fb_eib_kabinetFloorHeatingPowerSpRec(
	strData_Rec := fb_KL6301_0.str_Data_Rec,
	Group_Address := kabinetFloorHeatingPowerSp_adr,
	iData => kabinetFloorHeatingSp
	);
data2floor[103] := INT_TO_BYTE(kabinetFloorHeatingSp);

fb_eib_studioFloorHeatingPowerSpRec(
	strData_Rec := fb_KL6301_0.str_Data_Rec,
	Group_Address := studioFloorHeatingPowerSp_adr,
	iData => studioFloorHeatingSp
	);
data2floor[104] := INT_TO_BYTE(studioFloorHeatingSp);

fb_balkon_peryla_read(strData_Rec:=fb_KL6301_0.str_Data_Rec,   Group_Address:=balkon_peryla_adr);
IF NOT  fb_balkon_peryla_read.bDataReceive OR NOT fb_eib_twillight_rec.bDataReceive  THEN
	data2floor[100].0:= fb_balkon_peryla_read.bdata OR  fb_eib_twillight_rec.bData ;
END_IF
fb_kino_l_read(strData_Rec:=fb_KL6301_0.str_Data_Rec,   Group_Address:=kino_l_adr);
IF NOT  fb_kino_l_read.bDataReceive THEN
	data2floor[100].1:= fb_kino_l_read.bdata;
END_IF
fb_balkon_bra_read(strData_Rec:=fb_KL6301_0.str_Data_Rec,   Group_Address:=balkon_bra_adr);
IF NOT  fb_balkon_bra_read.bDataReceive OR NOT fb_eib_twillight_rec.bDataReceive THEN
	data2floor[100].2:= fb_balkon_bra_read.bdata OR fb_eib_twillight_rec.bData;
END_IF
fb_kabinet_balkon_l_read(strData_Rec:=fb_KL6301_0.str_Data_Rec,   Group_Address:=kabinet_balkon_l_adr);
IF NOT  fb_kabinet_balkon_l_read.bDataReceive THEN
	data2floor[100].3:= fb_kabinet_balkon_l_read.bdata;
END_IF
fb_balkon_read(strData_Rec:=fb_KL6301_0.str_Data_Rec,   Group_Address:=balkon_adr);
IF NOT  fb_balkon_read.bDataReceive THEN
	data2floor[100].4:= fb_balkon_read.bdata;
END_IF
fb_korydor1_read(strData_Rec:=fb_KL6301_0.str_Data_Rec,   Group_Address:=korydor1_adr);
IF NOT  fb_korydor1_read.bDataReceive THEN
	data2floor[100].5:= fb_korydor1_read.bdata;
END_IF
fb_kino_bra_read(strData_Rec:=fb_KL6301_0.str_Data_Rec,   Group_Address:=kino_bra_adr);
IF NOT  fb_kino_bra_read.bDataReceive THEN
	data2floor[100].6:= fb_kino_bra_read.bdata;
END_IF
fb_studio_pidsvitka_read(strData_Rec:=fb_KL6301_0.str_Data_Rec,   Group_Address:=studio_pidsvitka_adr);
IF NOT  fb_studio_pidsvitka_read.bDataReceive THEN
	data2floor[100].7:= fb_studio_pidsvitka_read.bdata;
END_IF
fb_skhody2_3_read(strData_Rec:=fb_KL6301_0.str_Data_Rec,   Group_Address:=skhody2_3_adr);
IF NOT  fb_skhody2_3_read.bDataReceive THEN
	data2floor[101].0:= fb_skhody2_3_read.bdata;
END_IF
fb_studio_l_read(strData_Rec:=fb_KL6301_0.str_Data_Rec,   Group_Address:=studio_l_adr);
IF NOT  fb_studio_l_read.bDataReceive THEN
	data2floor[101].1:= fb_studio_l_read.bdata;
END_IF
fb_kabinet_svitlo_read(strData_Rec:=fb_KL6301_0.str_Data_Rec,   Group_Address:=kabinet_svitlo_adr);
IF NOT  fb_kabinet_svitlo_read.bDataReceive THEN
	data2floor[101].2:= fb_kabinet_svitlo_read.bdata;
END_IF
fb_kabinet_kobra_read(strData_Rec:=fb_KL6301_0.str_Data_Rec,   Group_Address:=kabinet_kobra_adr);
IF NOT  fb_kabinet_kobra_read.bDataReceive THEN
	data2floor[101].3:= fb_kabinet_kobra_read.bdata;
END_IF
fb_tambur2_read(strData_Rec:=fb_KL6301_0.str_Data_Rec,   Group_Address:=tambur2_adr);
IF NOT  fb_tambur2_read.bDataReceive THEN
	data2floor[101].4:= fb_tambur2_read.bdata;
END_IF
fb_stend_read(strData_Rec:=fb_KL6301_0.str_Data_Rec,   Group_Address:=stend_adr);
IF NOT  fb_stend_read.bDataReceive THEN
	data2floor[101].5:= fb_stend_read.bdata;
END_IF
fb_skhody_peryla_read(strData_Rec:=fb_KL6301_0.str_Data_Rec,   Group_Address:=skhody_peryla_adr);
IF NOT  fb_skhody_peryla_read.bDataReceive OR NOT  fb_eib_twillight_rec.bDataReceive THEN
	data2floor[101].6:= fb_skhody_peryla_read.bdata OR  fb_eib_twillight_rec.bData;
END_IF

fb_kino_bra_dim_read(strData_Rec:=fb_KL6301_0.str_Data_Rec,   Group_Address:=kino_bra_dimming_adr);
IF NOT  fb_kino_bra_dim_read.bDataReceive THEN
	data2floor[102]:= INT_TO_BYTE(fb_kino_bra_dim_read.iData);
END_IF


(*sending*)
fb_balkon_peryla_send_status_ex(imode:=eib_send_mode_floor2, bStart:=eib_send_cyclical_start_floor2, str_Rec:=fb_KL6301_0.str_Data_Rec, bData:=balkon_peryla,  Group_Address:=balkon_peryla_status_adr);
fb_kino_l_send_status_ex(imode:=eib_send_mode_floor2, bStart:=eib_send_cyclical_start_floor2, str_Rec:=fb_KL6301_0.str_Data_Rec, bData:=kino_l,  Group_Address:=kino_l_status_adr);
fb_balkon_bra_send_status_ex(imode:=eib_send_mode_floor2, bStart:=eib_send_cyclical_start_floor2, str_Rec:=fb_KL6301_0.str_Data_Rec, bData:=balkon_bra,  Group_Address:=balkon_bra_status_adr);
fb_kabinet_balkon_l_send_status_ex(imode:=eib_send_mode_floor2, bStart:=eib_send_cyclical_start_floor2, str_Rec:=fb_KL6301_0.str_Data_Rec, bData:=kabinet_balkon_l,  Group_Address:=kabinet_balkon_l_status_adr);
fb_balkon_send_status_ex(imode:=eib_send_mode_floor2, bStart:=eib_send_cyclical_start_floor2, str_Rec:=fb_KL6301_0.str_Data_Rec, bData:=balkon,  Group_Address:=balkon_status_adr);
fb_korydor1_send_status_ex(imode:=eib_send_mode_floor2, bStart:=eib_send_cyclical_start_floor2, str_Rec:=fb_KL6301_0.str_Data_Rec, bData:=korydor1,  Group_Address:=korydor1_status_adr);
fb_kino_bra_send_status_ex(imode:=eib_send_mode_floor2, bStart:=eib_send_cyclical_start_floor2, str_Rec:=fb_KL6301_0.str_Data_Rec, bData:=kino_bra,  Group_Address:=kino_bra_status_adr);
fb_studio_pidsvitka_send_status_ex(imode:=eib_send_mode_floor2, bStart:=eib_send_cyclical_start_floor2, str_Rec:=fb_KL6301_0.str_Data_Rec, bData:=studio_pidsvitka,  Group_Address:=studio_pidsvitka_status_adr);
fb_skhody2_3_send_status_ex(imode:=eib_send_mode_floor2, bStart:=eib_send_cyclical_start_floor2, str_Rec:=fb_KL6301_0.str_Data_Rec, bData:=skhody2_3,  Group_Address:=skhody2_3_status_adr);
fb_studio_l_send_status_ex(imode:=eib_send_mode_floor2, bStart:=eib_send_cyclical_start_floor2, str_Rec:=fb_KL6301_0.str_Data_Rec, bData:=studio_l,  Group_Address:=studio_l_status_adr);
fb_kabinet_svitlo_send_status_ex(imode:=eib_send_mode_floor2, bStart:=eib_send_cyclical_start_floor2, str_Rec:=fb_KL6301_0.str_Data_Rec, bData:=kabinet_svitlo,  Group_Address:=kabinet_svitlo_status_adr);
fb_kabinet_kobra_send_status_ex(imode:=eib_send_mode_floor2, bStart:=eib_send_cyclical_start_floor2, str_Rec:=fb_KL6301_0.str_Data_Rec, bData:=kabinet_kobra,  Group_Address:=kabinet_kobra_status_adr);
fb_tambur2_send_status_ex(imode:=eib_send_mode_floor2, bStart:=eib_send_cyclical_start_floor2, str_Rec:=fb_KL6301_0.str_Data_Rec, bData:=tambur2,  Group_Address:=tambur2_status_adr);
fb_stend_send_status_ex(imode:=eib_send_mode_floor2, bStart:=eib_send_cyclical_start_floor2, str_Rec:=fb_KL6301_0.str_Data_Rec, bData:=stend,  Group_Address:=stend_status_adr);
fb_skhody_peryla_send_status_ex(imode:=eib_send_mode_floor2, bStart:=eib_send_cyclical_start_floor2, str_Rec:=fb_KL6301_0.str_Data_Rec, bData:=skhody_peryla,  Group_Address:=skhody_peryla_status_adr);
fb_kino_bra_send_dim_status_ex(imode:=eib_send_mode_floor2, bstart:=eib_send_cyclical_start_floor2, str_Rec:=fb_KL6301_0.str_Data_Rec, idata:=BYTE_TO_INT(kino_bra_dim_value) );


IF fb_balkon_peryla_send_status_ex.bBusy THEN
	data2floor[100].0:=balkon_peryla;
END_IF
IF fb_kino_l_send_status_ex.bBusy OR fb_heartbeat_timer.Q THEN
	data2floor[100].1:=kino_l;
END_IF
IF fb_balkon_bra_send_status_ex.bBusy OR fb_heartbeat_timer.Q THEN
	data2floor[100].2:=balkon_bra;
END_IF
IF fb_kabinet_balkon_l_send_status_ex.bBusy OR fb_heartbeat_timer.Q THEN
	data2floor[100].3:=kabinet_balkon_l;
END_IF
IF fb_balkon_send_status_ex.bBusy OR fb_heartbeat_timer.Q THEN
	data2floor[100].4:=balkon;
END_IF
IF fb_korydor1_send_status_ex.bBusy OR fb_heartbeat_timer.Q THEN
	data2floor[100].5:=korydor1;
END_IF
IF fb_kino_bra_send_status_ex.bBusy OR fb_heartbeat_timer.Q THEN
	data2floor[100].6:=kino_bra;
END_IF
IF fb_studio_pidsvitka_send_status_ex.bBusy OR fb_heartbeat_timer.Q THEN
	data2floor[100].7:=studio_pidsvitka;
END_IF
IF fb_skhody2_3_send_status_ex.bBusy OR fb_heartbeat_timer.Q THEN
	data2floor[101].0:=skhody2_3;
END_IF
IF fb_studio_l_send_status_ex.bBusy OR fb_heartbeat_timer.Q THEN
	data2floor[101].1:=studio_l;
END_IF
IF fb_kabinet_svitlo_send_status_ex.bBusy OR fb_heartbeat_timer.Q THEN
	data2floor[101].2:=kabinet_svitlo;
END_IF
IF fb_kabinet_kobra_send_status_ex.bBusy OR fb_heartbeat_timer.Q THEN
	data2floor[101].3:=kabinet_kobra;
END_IF
IF fb_tambur2_send_status_ex.bBusy OR fb_heartbeat_timer.Q THEN
	data2floor[101].4:=tambur2;
END_IF
IF fb_stend_send_status_ex.bBusy OR fb_heartbeat_timer.Q THEN
	data2floor[101].5:=stend;
END_IF
IF fb_skhody_peryla_send_status_ex.bBusy OR fb_heartbeat_timer.Q THEN
	data2floor[101].6:=skhody_peryla;
END_IF
IF fb_kino_bra_send_dim_status_ex.bBusy THEN
	data2floor[102]:=INT_TO_BYTE(kino_bra_dim_value);
END_IF
END_ACTION
ACTION floor3:
(*read*)
fb_spalnya_kontrazhury_read(
	strData_Rec := fb_KL6301_0.str_Data_Rec,
	Group_Address := spalnya_kontrazhury_adr,
	bData => eib_spalnya_kontrazhury
	);

fb_spalnya_balkon_read(
	strData_Rec := fb_KL6301_0.str_Data_Rec,
	Group_Address := spalnya_balkon_adr,
	bData => eib_spalnya_balkon
	);

fb_spalnya_kulbaba_read(
	strData_Rec := fb_KL6301_0.str_Data_Rec,
	Group_Address := spalnya_kulbaba_adr,
	bData => eib_spalnya_kulbaba
	);

fb_eib_su3FloorHeatingPowerSpRec(
	strData_Rec := fb_KL6301_0.str_Data_Rec,
	Group_Address := su3FloorHeatingPowerSp_adr,
	iData => su3FloorHeatingSp
	);

fb_eib_freshbarFloorHeatingPowerSpRec(
	strData_Rec := fb_KL6301_0.str_Data_Rec,
	Group_Address := freshbarFloorHeatingPowerSp_adr,
	iData => freshbarFloorHeatingSp
	);

fb_eib_servernaFloorHeatingPowerSpRec(
	strData_Rec := fb_KL6301_0.str_Data_Rec,
	Group_Address := servernaFloorHeatingPowerSp_adr,
	iData => servernaFloorHeatingSp
	);

fb_eib_spalnyaFloorHeatingPowerSpRec(
	strData_Rec := fb_KL6301_0.str_Data_Rec,
	Group_Address := spalnyaFloorHeatingPowerSp_adr,
	iData => spalnyaFloorHeatingSp
	);

fb_eib_dytjachaFloorHeatingPowerSpRec(
	strData_Rec := fb_KL6301_0.str_Data_Rec,
	Group_Address := dytjachaFloorHeatingPowerSp_adr,
	iData => dytjachaFloorHeatingSp
	);

(*
fb_spalnya_kontrazhur_b_read(strData_Rec:=fb_KL6301_0.str_Data_Rec, Group_Address:=spalnya_kontrazhur_b_adr);
fb_spalnya_kontrazhur_l_read(strData_Rec:=fb_KL6301_0.str_Data_Rec, Group_Address:=spalnya_kontrazhur_l_adr);
*)
fb_su3_stina_read(
	strData_Rec := fb_KL6301_0.str_Data_Rec,
	Group_Address := su3_stina_adr,
	bData => eib_su3_stina
	);

fb_su3_pidsvitka_read(
	strData_Rec := fb_KL6301_0.str_Data_Rec,
	Group_Address := su3_pidsvitka_adr,
	bData => eib_su3_pidsvitka
	);

fb_su3_bra_read(
	strData_Rec := fb_KL6301_0.str_Data_Rec,
	Group_Address := su3_bra_adr,
	bData => eib_su3_bra
	);

fb_su3_kontrazhur_read(
	strData_Rec := fb_KL6301_0.str_Data_Rec,
	Group_Address := su3_kontrazhury_adr,
	bData => eib_su3_kontrazhury
	);

fb_su3_vent_read(
	strData_Rec := fb_KL6301_0.str_Data_Rec,
	Group_Address := su3_vent_adr,
	bData => eib_su3_vent
	);

fb_su3_lampa_read(
	strData_Rec := fb_KL6301_0.str_Data_Rec,
	Group_Address := su3_lampa_adr,
	bData => eib_su3_lampa
	);

fb_dytjacha_read(
	strData_Rec := fb_KL6301_0.str_Data_Rec,
	Group_Address := dytjacha_adr,
	bData => eib_dytjacha
	);

fb_dytjacha_bra_read(
	strData_Rec := fb_KL6301_0.str_Data_Rec,
	Group_Address := dytjacha_bra_adr,
	bData => eib_dytjacha_bra
	);

fb_garderob_read(
	strData_Rec := fb_KL6301_0.str_Data_Rec,
	Group_Address := garderob_adr,
	bData => eib_garderob
	);

fb_bar_read(
	strData_Rec := fb_KL6301_0.str_Data_Rec,
	Group_Address := bar_adr,
	bData => eib_bar
	);

fb_korydor_skeli_read(
	strData_Rec := fb_KL6301_0.str_Data_Rec,
	Group_Address := korydor_skeli_adr,
	bData => eib_korydor_skeli
	);

fb_choven_read(
	strData_Rec := fb_KL6301_0.str_Data_Rec,
	Group_Address := choven_adr,
	bData => eib_choven
	);

fb_korydor_lampa_read(
	strData_Rec := fb_KL6301_0.str_Data_Rec,
	Group_Address := korydor_lampa_adr,
	bData => eib_korydor_lampa
	);

fb_serverna_read(
	strData_Rec := fb_KL6301_0.str_Data_Rec,
	Group_Address := serverna_adr,
	bData => eib_serverna
	);

fb_korydor_svitlo_read(
	strData_Rec := fb_KL6301_0.str_Data_Rec,
	Group_Address := korydor_svitlo_adr,
	bData => eib_korydor_svitlo
	);

(*sending*)
(*
fb_spalnya_kontrazhur_b_send_status_ex(imode:=eib_send_mode_floor3, bStart:=eib_send_cyclical_start_floor3, str_Rec:=fb_KL6301_0.str_Data_Rec, Group_Address:=spalnya_kontrazhur_b_status_adr, bData:=spalnya_kontrazhur_b);
fb_spalnya_kontrazhur_l_send_status_ex(imode:=eib_send_mode_floor3, bStart:=eib_send_cyclical_start_floor3, str_Rec:=fb_KL6301_0.str_Data_Rec, Group_Address:=spalnya_kontrazhur_l_status_adr, bData:=spalnya_kontrazhur_l);

*)
fb_su3_stina_send_status_ex(
	imode := eib_send_mode_floor3,
	bStart := eib_send_cyclical_start_floor3,
	str_Rec := fb_KL6301_0.str_Data_Rec,
	Group_Address := su3_stina_status_adr,
	bData := su3_stina
	);

fb_su3_pidsvitka_send_status_ex(
	imode := eib_send_mode_floor3,
	bStart := eib_send_cyclical_start_floor3,
	str_Rec := fb_KL6301_0.str_Data_Rec,
	Group_Address := su3_pidsvitka_status_adr,
	bData := su3_pidsvitka
	);

fb_su3_bra_send_status_ex(
	imode := eib_send_mode_floor3,
	bStart := eib_send_cyclical_start_floor3,
	str_Rec := fb_KL6301_0.str_Data_Rec,
	Group_Address := su3_bra_status_adr,
	bData := su3_bra
	);

fb_su3_kontrazhur_send_status_ex(
	imode := eib_send_mode_floor3,
	bStart := eib_send_cyclical_start_floor3,
	str_Rec := fb_KL6301_0.str_Data_Rec,
	Group_Address := su3_kontrazhury_status_adr,
	bData := su3_kontrazhur
	);

fb_su3_vent_send_status_ex(
	imode := eib_send_mode_floor3,
	bStart := eib_send_cyclical_start_floor3,
	str_Rec := fb_KL6301_0.str_Data_Rec,
	Group_Address := su3_vent_status_adr,
	bData := su3_vent
	);

fb_su3_lampa_send_status_ex(
	imode := eib_send_mode_floor3,
	bStart := eib_send_cyclical_start_floor3,
	str_Rec := fb_KL6301_0.str_Data_Rec,
	Group_Address := su3_lampa_status_adr,
	bData := su3_lampa
	);

fb_dytjacha_send_status_ex(
	imode := eib_send_mode_floor3,
	bStart := eib_send_cyclical_start_floor3,
	str_Rec := fb_KL6301_0.str_Data_Rec,
	Group_Address := dytjacha_status_adr,
	bData := dytjacha
	);

fb_dytjacha_bra_send_status_ex(
	imode := eib_send_mode_floor3,
	bStart := eib_send_cyclical_start_floor3,
	str_Rec := fb_KL6301_0.str_Data_Rec,
	Group_Address := dytjacha_bra_status_adr,
	bData := dytjacha_bra
	);

fb_garderob_send_status_ex(
	imode := eib_send_mode_floor3,
	bStart := eib_send_cyclical_start_floor3,
	str_Rec := fb_KL6301_0.str_Data_Rec,
	Group_Address := garderob_status_adr,
	bData := garderob
	);

fb_bar_send_status_ex(
	imode := eib_send_mode_floor3,
	bStart := eib_send_cyclical_start_floor3,
	str_Rec := fb_KL6301_0.str_Data_Rec,
	Group_Address := bar_status_adr,
	bData := bar
	);

fb_korydor_skeli_send_status_ex(
	imode := eib_send_mode_floor3,
	bStart := eib_send_cyclical_start_floor3,
	str_Rec := fb_KL6301_0.str_Data_Rec,
	Group_Address := korydor_skeli_status_adr,
	bData := korydor_skeli
	);

fb_choven_send_status_ex(
	imode := eib_send_mode_floor3,
	bStart := eib_send_cyclical_start_floor3,
	str_Rec := fb_KL6301_0.str_Data_Rec,
	Group_Address := choven_status_adr,
	bData := choven
	);

fb_korydor_lampa_send_status_ex(
	imode := eib_send_mode_floor3,
	bStart := eib_send_cyclical_start_floor3,
	str_Rec := fb_KL6301_0.str_Data_Rec,
	Group_Address := korydor_lampa_status_adr,
	bData := korydor_lampa
	);

fb_serverna_send_status_ex(
	imode := eib_send_mode_floor3,
	bStart := eib_send_cyclical_start_floor3,
	str_Rec := fb_KL6301_0.str_Data_Rec,
	Group_Address := serverna_status_adr,
	bData := serverna
	);

fb_korydor_svitlo_send_status_ex(
	imode := eib_send_mode_floor3,
	bStart := eib_send_cyclical_start_floor3,
	str_Rec := fb_KL6301_0.str_Data_Rec,
	Group_Address := korydor_svitlo_status_adr,
	bData := korydor_svitlo
	);

fb_spalnya_balkon_send_status_ex(
	imode := eib_send_mode_floor3,
	bStart := eib_send_cyclical_start_floor3,
	str_Rec := fb_KL6301_0.str_Data_Rec,
	Group_Address := spalnya_balkon_status_adr,
	bData := spalnya_balkon
	);

fb_spalnya_kulbaba_send_status_ex(
	imode := eib_send_mode_floor3,
	bStart := eib_send_cyclical_start_floor3,
	str_Rec := fb_KL6301_0.str_Data_Rec,
	Group_Address := spalnya_kulbaba_status_adr,
	bData := spalnya_kulbaba
	);

fb_spalnya_kontrazhury_send_status_ex(
	imode := eib_send_mode_floor3,
	bStart := eib_send_cyclical_start_floor3,
	str_Rec := fb_KL6301_0.str_Data_Rec,
	Group_Address := spalnya_kontrazhury_status_adr,
	bData :=spalnya_kontrazhur
	);

fb_spalnya_lift_send_status_ex(
	imode := eib_send_mode_floor3,
	bStart := eib_send_cyclical_start_floor3,
	str_Rec := fb_KL6301_0.str_Data_Rec,
	Group_Address := lift_spalnya_status_EIB_addr,
	bData := eib_lift_spalnya_move
	);
END_ACTION
ACTION gym_and_outside:
data_gym[0].0:=bDarkOutside OR b_eib_twillight;
data_gym[0].1:=1;

data_gym[1]:=WORD_TO_BYTE(system_time.wHour);
data_gym[3]:=WORD_TO_BYTE(system_time.wMinute);

MEMCPY(ADR(data_gym[6] ), ADR(OAT), SIZEOF(OAT));


fb_outside_bigBulbs_read(strData_Rec:=fb_KL6301_0.str_Data_Rec, Group_Address:=outside_bigBulbs_adr );
IF NOT  fb_outside_Bigbulbs_read.bDataReceive THEN
	data_gym[12].3:= fb_outside_bigBulbs_read.bdata;
END_IF

fb_outside_pingPongTable_read(strData_Rec:=fb_KL6301_0.str_Data_Rec, Group_Address:=outside_pingPongTable_adr );
IF NOT  fb_outside_pingPongTable_read.bDataReceive THEN
	data_gym[12].4:= fb_outside_pingPongTable_read.bdata;
END_IF
fb_outside_plantsLightning_read(strData_Rec:=fb_KL6301_0.str_Data_Rec, Group_Address:=outside_plantsLightning_adr );
IF NOT  fb_outside_plantsLightning_read.bDataReceive THEN
	data_gym[12].5:= fb_outside_plantsLightning_read.bdata;
END_IF

fb_outside_smallBulbs_read(strData_Rec:=fb_KL6301_0.str_Data_Rec, Group_Address:=outside_smallBulbs_adr );
IF NOT  fb_outside_smallBulbs_read.bDataReceive THEN
	data_gym[12].6:= fb_outside_smallBulbs_read.bdata;
END_IF


(*sending*)


fb_outside_bigBulbs_send_status_ex(imode:=eib_send_mode_floor4, bStart:=eib_send_cyclical_start_floor4, str_Rec:=fb_KL6301_0.str_Data_Rec, bData:=outside_bigBulbs,  Group_Address:=outside_bigBulbs_status_adr);
fb_outside_pingPongTable_send_status_ex(imode:=eib_send_mode_floor4, bStart:=eib_send_cyclical_start_floor4, str_Rec:=fb_KL6301_0.str_Data_Rec, bData:=outside_pingPongTable,  Group_Address:=outside_pingPongTable_status_adr);
fb_outside_plantsLightning_send_status_ex(imode:=eib_send_mode_floor4, bStart:=eib_send_cyclical_start_floor4, str_Rec:=fb_KL6301_0.str_Data_Rec, bData:=outside_plantsLightning,  Group_Address:=outside_plantsLightning_status_adr);
fb_outside_smallBulbs_send_status_ex(imode:=eib_send_mode_floor4, bStart:=eib_send_cyclical_start_floor4, str_Rec:=fb_KL6301_0.str_Data_Rec, bData:=outside_smallBulbs,  Group_Address:=outside_smallBulbs_status_adr);


IF fb_gym_light_send_status_ex.bBusy OR fb_heartbeat_timer.Q  THEN
	data_gym[12].2:=gym_light;
END_IF


IF fb_outside_bigBulbs_send_status_ex.bBusy OR fb_heartbeat_timer.Q  THEN
	data_gym[12].3:=outside_bigBulbs;
END_IF

IF fb_outside_pingPongTable_send_status_ex.bBusy OR fb_heartbeat_timer.Q  THEN
	data_gym[12].4:=outside_pingPongTable;
END_IF

IF fb_outside_plantsLightning_send_status_ex.bBusy OR fb_heartbeat_timer.Q  THEN
	data_gym[12].5:=outside_plantsLightning;
END_IF

IF fb_outside_smallBulbs_send_status_ex.bBusy OR fb_heartbeat_timer.Q  THEN
	data_gym[12].6:=outside_smallBulbs;
END_IF
END_ACTION
ACTION timers:
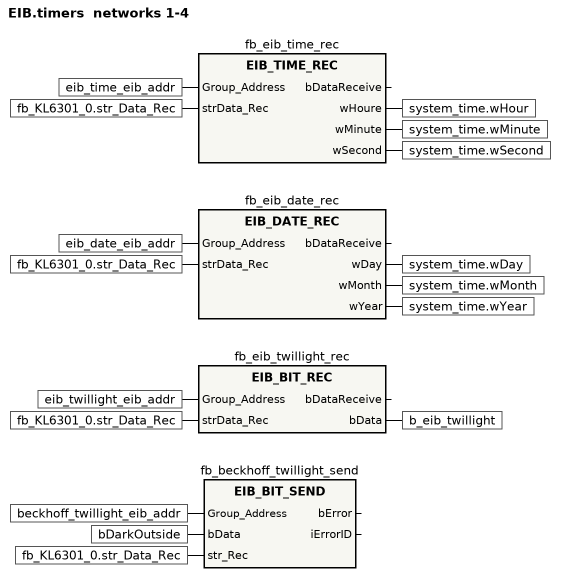
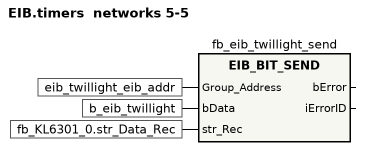
_FBD_ (* Function Block Diagram *)
NETWORK 1
	fb_eib_time_rec:EIB_TIME_REC(Group_Address: eib_time_eib_addr, strData_Rec: fb_KL6301_0.str_Data_Rec, wHoure => system_time.wHour, wMinute => system_time.wMinute, wSecond => system_time.wSecond)
NETWORK 2
	fb_eib_date_rec:EIB_DATE_REC(Group_Address: eib_date_eib_addr, strData_Rec: fb_KL6301_0.str_Data_Rec, wDay => system_time.wDay, wMonth => system_time.wMonth, wYear => system_time.wYear)
NETWORK 3
	fb_eib_twillight_rec:EIB_BIT_REC(Group_Address: eib_twillight_eib_addr, strData_Rec: fb_KL6301_0.str_Data_Rec, bData => b_eib_twillight)
NETWORK 4
	fb_beckhoff_twillight_send:EIB_BIT_SEND(Group_Address: beckhoff_twillight_eib_addr, bData: bDarkOutside, str_Rec: fb_KL6301_0.str_Data_Rec)
NETWORK 5
	fb_eib_twillight_send:EIB_BIT_SEND(Group_Address: eib_twillight_eib_addr, bData: b_eib_twillight, str_Rec: fb_KL6301_0.str_Data_Rec)
_END_FBD_
(* the same logic as Structured Text *)
(* Network 1 *)
fb_eib_time_rec(Group_Address := eib_time_eib_addr, strData_Rec := fb_KL6301_0.str_Data_Rec);
system_time.wHour := fb_eib_time_rec.wHoure;
system_time.wMinute := fb_eib_time_rec.wMinute;
system_time.wSecond := fb_eib_time_rec.wSecond;
(* Network 2 *)
fb_eib_date_rec(Group_Address := eib_date_eib_addr, strData_Rec := fb_KL6301_0.str_Data_Rec);
system_time.wDay := fb_eib_date_rec.wDay;
system_time.wMonth := fb_eib_date_rec.wMonth;
system_time.wYear := fb_eib_date_rec.wYear;
(* Network 3 *)
fb_eib_twillight_rec(Group_Address := eib_twillight_eib_addr, strData_Rec := fb_KL6301_0.str_Data_Rec);
b_eib_twillight := fb_eib_twillight_rec.bData;
(* Network 4 *)
fb_beckhoff_twillight_send(Group_Address := beckhoff_twillight_eib_addr, bData := bDarkOutside, str_Rec := fb_KL6301_0.str_Data_Rec);
(* Network 5 *)
fb_eib_twillight_send(Group_Address := eib_twillight_eib_addr, bData := b_eib_twillight, str_Rec := fb_KL6301_0.str_Data_Rec);
END_ACTION

(* POU RANGE_TO_RANGE, ST *)
FUNCTION RANGE_TO_RANGE : INT
VAR_INPUT
	by_input:BYTE;
	in_low_value: INT;
	in_high_value:INT;
	out_low_value: INT;
	out_high_value:INT;
END_VAR
VAR
	r_res: REAL;
	r_input: REAL;
END_VAR
r_input:=BYTE_TO_REAL(by_input);
IF out_high_value>out_low_value THEN
	r_res:=r_input/(in_high_value - in_low_value)*(out_high_value - out_low_value);
ELSE
	r_res:=out_low_value - (r_input / (in_high_value - in_low_value)*(out_low_value - out_high_value));
END_IF
RANGE_TO_RANGE:=REAL_TO_INT(r_res);
END_FUNCTION

(* POU GREATEST_OF, ST *)
FUNCTION GREATEST_OF : REAL
VAR_INPUT
	r_in1,r_in2:REAL;
END_VAR
VAR
END_VAR
IF r_in1>=r_in2 THEN
	GREATEST_OF:=r_in1;
ELSE
	GREATEST_OF:=r_in2;
END_IF
END_FUNCTION

(* POU Light, CFC *)
PROGRAM Light
VAR
	fbSpalnya_kontrazhury: FB_Light;
	fbSpalnya_balkon: FB_Light;
	fbSpalnya_light: FB_Light;
	fbSu3_vent: fbMoovingSensorLight;
	fbSu3_stina: FB_Light;
	fbSu3_bra: FB_Light;
	fbSu3_lampa: FB_Light;
	fbSu3_pidsvitka: FB_Light;
	fbDytjacha: FB_Light;
	fbDytjacha_bra: FB_Light;
	fbGarderob: FB_Light;
	fbServerna: FB_Light;
	fbBar: FB_Light;
	fbChoven:fbMoovingSensorLight;
	fbKorydor_skeli: fbMoovingSensorLight;
	fbKorydor_svitlo:fbMoovingSensorLight;
	fbKorydor_lampa:fbMoovingSensorLight;
	fbSu3_1_sw:				FB_ShortLongClick;
	fbSu3_2_sw:				FB_ShortLongClick;
	fbSpalnya_1_sw:			FB_ShortLongClick;
	fbSpalnya_2_sw:			FB_ShortLongClick;
	tambur3_2_short_click:BOOL;
	tambur3_2_long_click:BOOL;
	tambur3_2_short_click_TP:TP;
	tambur3_2_long_click_TP:TP;

	longPressDelay: TIME:=t#500ms;
	lightDuration:TIME:=t#2m;




	fbShtorySpalnya: FB_VenetianBlindEx1Switch;
	fbTulSpalnya: FB_VenetianBlindEx1Switch;

	fbTambur3_2_sw: FB_ShortLongClick;
	fbSpalnyaLift: FB_RoofWindow;
	fbEIB_lift_spalnya_status_SET_RESET: SEMA;
END_VAR
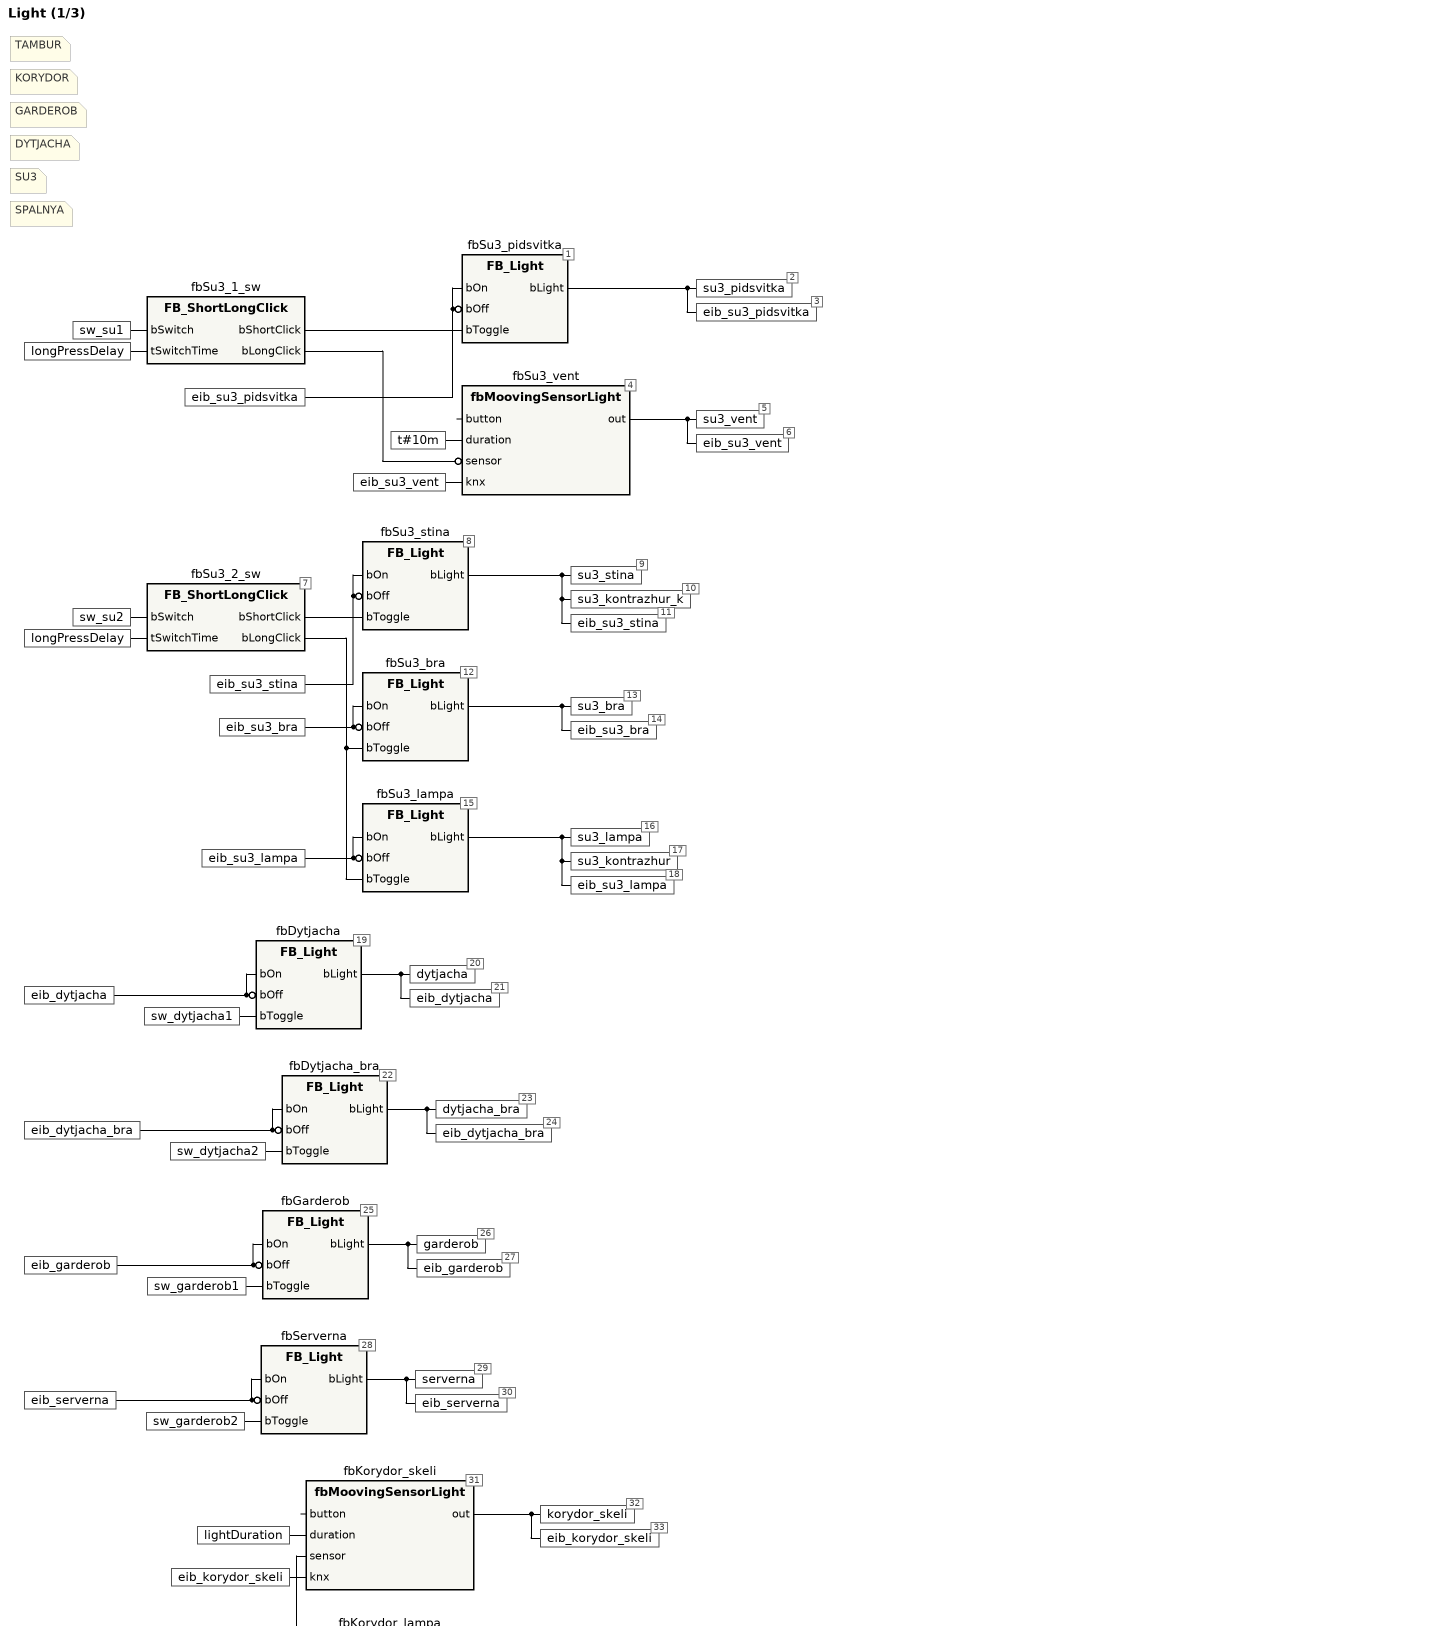
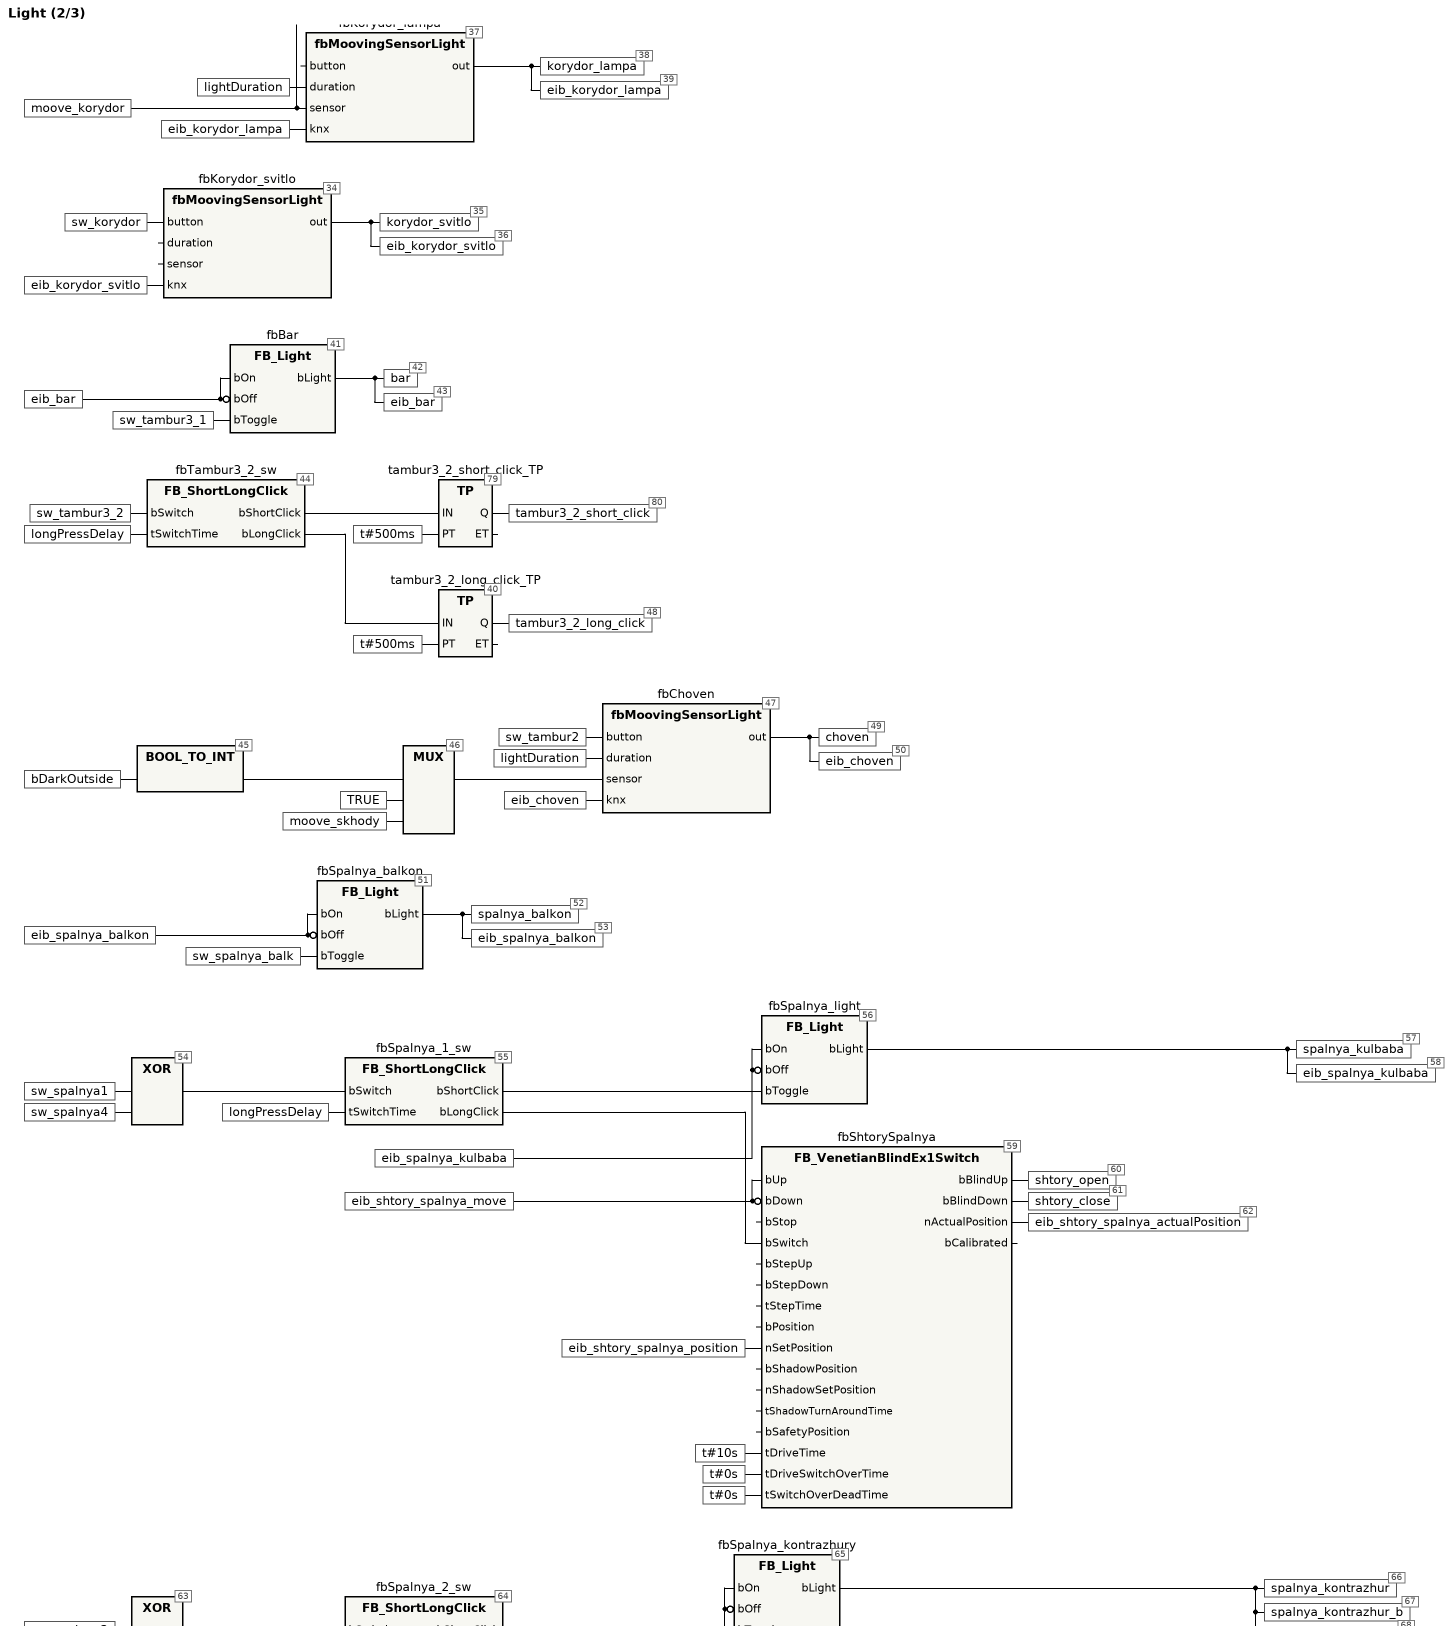
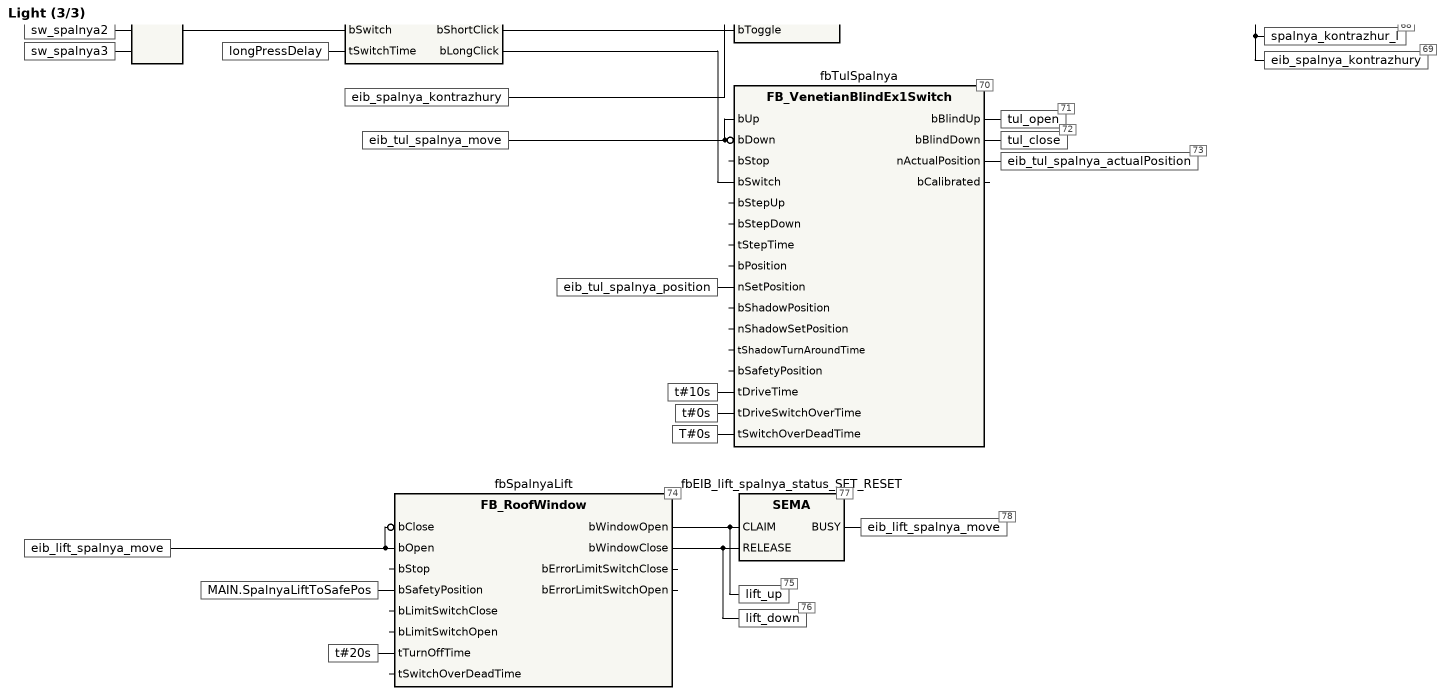
_CFC_ (* Continuous Function Chart, elements in execution order *)
(* TAMBUR *)
(* KORYDOR *)
(* GARDEROB *)
(* DYTJACHA *)
(* SU3 *)
(* SPALNYA *)
#0 fbSu3_1_sw:FB_ShortLongClick(bSwitch: sw_su1, tSwitchTime: longPressDelay)
#1 fbSu3_pidsvitka:FB_Light(bOn: eib_su3_pidsvitka, bOff: NOT eib_su3_pidsvitka, bToggle: #0.bShortClick)
#2 su3_pidsvitka <= #1.bLight
#3 eib_su3_pidsvitka <= #1.bLight
#4 fbSu3_vent:fbMoovingSensorLight(button: -, duration: t#10m, sensor: NOT #0.bLongClick, knx: eib_su3_vent)
#5 su3_vent <= #4.out
#6 eib_su3_vent <= #4.out
#7 fbSu3_2_sw:FB_ShortLongClick(bSwitch: sw_su2, tSwitchTime: longPressDelay)
#8 fbSu3_stina:FB_Light(bOn: eib_su3_stina, bOff: NOT eib_su3_stina, bToggle: #7.bShortClick)
#9 su3_stina <= #8.bLight
#10 su3_kontrazhur_k <= #8.bLight
#11 eib_su3_stina <= #8.bLight
#12 fbSu3_bra:FB_Light(bOn: eib_su3_bra, bOff: NOT eib_su3_bra, bToggle: #7.bLongClick)
#13 su3_bra <= #12.bLight
#14 eib_su3_bra <= #12.bLight
#15 fbSu3_lampa:FB_Light(bOn: eib_su3_lampa, bOff: NOT eib_su3_lampa, bToggle: #7.bLongClick)
#16 su3_lampa <= #15.bLight
#17 su3_kontrazhur <= #15.bLight
#18 eib_su3_lampa <= #15.bLight
#19 fbDytjacha:FB_Light(bOn: eib_dytjacha, bOff: NOT eib_dytjacha, bToggle: sw_dytjacha1)
#20 dytjacha <= #19.bLight
#21 eib_dytjacha <= #19.bLight
#22 fbDytjacha_bra:FB_Light(bOn: eib_dytjacha_bra, bOff: NOT eib_dytjacha_bra, bToggle: sw_dytjacha2)
#23 dytjacha_bra <= #22.bLight
#24 eib_dytjacha_bra <= #22.bLight
#25 fbGarderob:FB_Light(bOn: eib_garderob, bOff: NOT eib_garderob, bToggle: sw_garderob1)
#26 garderob <= #25.bLight
#27 eib_garderob <= #25.bLight
#28 fbServerna:FB_Light(bOn: eib_serverna, bOff: NOT eib_serverna, bToggle: sw_garderob2)
#29 serverna <= #28.bLight
#30 eib_serverna <= #28.bLight
#31 fbKorydor_skeli:fbMoovingSensorLight(button: -, duration: lightDuration, sensor: moove_korydor, knx: eib_korydor_skeli)
#32 korydor_skeli <= #31.out
#33 eib_korydor_skeli <= #31.out
#34 fbKorydor_svitlo:fbMoovingSensorLight(button: sw_korydor, duration: -, sensor: -, knx: eib_korydor_svitlo)
#35 korydor_svitlo <= #34.out
#36 eib_korydor_svitlo <= #34.out
#37 fbKorydor_lampa:fbMoovingSensorLight(button: -, duration: lightDuration, sensor: moove_korydor, knx: eib_korydor_lampa)
#38 korydor_lampa <= #37.out
#39 eib_korydor_lampa <= #37.out
#40 tambur3_2_long_click_TP:TP(IN: #44.bLongClick, PT: t#500ms)
#41 fbBar:FB_Light(bOn: eib_bar, bOff: NOT eib_bar, bToggle: sw_tambur3_1)
#42 bar <= #41.bLight
#43 eib_bar <= #41.bLight
#44 fbTambur3_2_sw:FB_ShortLongClick(bSwitch: sw_tambur3_2, tSwitchTime: longPressDelay)
#45 BOOL_TO_INT(bDarkOutside)
#46 MUX(#45, TRUE, moove_skhody)
#47 fbChoven:fbMoovingSensorLight(button: sw_tambur2, duration: lightDuration, sensor: #46, knx: eib_choven)
#48 tambur3_2_long_click <= #40.Q
#49 choven <= #47.out
#50 eib_choven <= #47.out
#51 fbSpalnya_balkon:FB_Light(bOn: eib_spalnya_balkon, bOff: NOT eib_spalnya_balkon, bToggle: sw_spalnya_balk)
#52 spalnya_balkon <= #51.bLight
#53 eib_spalnya_balkon <= #51.bLight
#54 XOR(sw_spalnya1, sw_spalnya4)
#55 fbSpalnya_1_sw:FB_ShortLongClick(bSwitch: #54, tSwitchTime: longPressDelay)
#56 fbSpalnya_light:FB_Light(bOn: eib_spalnya_kulbaba, bOff: NOT eib_spalnya_kulbaba, bToggle: #55.bShortClick)
#57 spalnya_kulbaba <= #56.bLight
#58 eib_spalnya_kulbaba <= #56.bLight
#59 fbShtorySpalnya:FB_VenetianBlindEx1Switch(bUp: eib_shtory_spalnya_move, bDown: NOT eib_shtory_spalnya_move, bStop: -, bSwitch: #55.bLongClick, bStepUp: -, bStepDown: -, tStepTime: -, bPosition: -, nSetPosition: eib_shtory_spalnya_position, bShadowPosition: -, nShadowSetPosition: -, tShadowTurnAroundTime: -, bSafetyPosition: -, tDriveTime: t#10s, tDriveSwitchOverTime: t#0s, tSwitchOverDeadTime: t#0s)
#60 shtory_open <= #59.bBlindUp
#61 shtory_close <= #59.bBlindDown
#62 eib_shtory_spalnya_actualPosition <= #59.nActualPosition
#63 XOR(sw_spalnya2, sw_spalnya3)
#64 fbSpalnya_2_sw:FB_ShortLongClick(bSwitch: #63, tSwitchTime: longPressDelay)
#65 fbSpalnya_kontrazhury:FB_Light(bOn: eib_spalnya_kontrazhury, bOff: NOT eib_spalnya_kontrazhury, bToggle: #64.bShortClick)
#66 spalnya_kontrazhur <= #65.bLight
#67 spalnya_kontrazhur_b <= #65.bLight
#68 spalnya_kontrazhur_l <= #65.bLight
#69 eib_spalnya_kontrazhury <= #65.bLight
#70 fbTulSpalnya:FB_VenetianBlindEx1Switch(bUp: eib_tul_spalnya_move, bDown: NOT eib_tul_spalnya_move, bStop: -, bSwitch: #64.bLongClick, bStepUp: -, bStepDown: -, tStepTime: -, bPosition: -, nSetPosition: eib_tul_spalnya_position, bShadowPosition: -, nShadowSetPosition: -, tShadowTurnAroundTime: -, bSafetyPosition: -, tDriveTime: t#10s, tDriveSwitchOverTime: t#0s, tSwitchOverDeadTime: T#0s)
#71 tul_open <= #70.bBlindUp
#72 tul_close <= #70.bBlindDown
#73 eib_tul_spalnya_actualPosition <= #70.nActualPosition
#74 fbSpalnyaLift:FB_RoofWindow(bClose: NOT eib_lift_spalnya_move, bOpen: eib_lift_spalnya_move, bStop: -, bSafetyPosition: MAIN.SpalnyaLiftToSafePos, bLimitSwitchClose: -, bLimitSwitchOpen: -, tTurnOffTime: t#20s, tSwitchOverDeadTime: -)
#75 lift_up <= #74.bWindowOpen
#76 lift_down <= #74.bWindowClose
#77 fbEIB_lift_spalnya_status_SET_RESET:SEMA(CLAIM: #74.bWindowOpen, RELEASE: #74.bWindowClose)
#78 eib_lift_spalnya_move <= #77.BUSY
#79 tambur3_2_short_click_TP:TP(IN: #44.bShortClick, PT: t#500ms)
#80 tambur3_2_short_click <= #79.Q
_END_CFC_
(* the same logic as Structured Text *)
(* TAMBUR *)
(* KORYDOR *)
(* GARDEROB *)
(* DYTJACHA *)
(* SU3 *)
(* SPALNYA *)
fbSu3_1_sw(bSwitch := sw_su1, tSwitchTime := longPressDelay);
fbSu3_pidsvitka(bOn := eib_su3_pidsvitka, bOff := NOT eib_su3_pidsvitka, bToggle := fbSu3_1_sw.bShortClick);
su3_pidsvitka := fbSu3_pidsvitka.bLight;
eib_su3_pidsvitka := fbSu3_pidsvitka.bLight;
fbSu3_vent(duration := t#10m, sensor := NOT fbSu3_1_sw.bLongClick, knx := eib_su3_vent);
su3_vent := fbSu3_vent.out;
eib_su3_vent := fbSu3_vent.out;
fbSu3_2_sw(bSwitch := sw_su2, tSwitchTime := longPressDelay);
fbSu3_stina(bOn := eib_su3_stina, bOff := NOT eib_su3_stina, bToggle := fbSu3_2_sw.bShortClick);
su3_stina := fbSu3_stina.bLight;
su3_kontrazhur_k := fbSu3_stina.bLight;
eib_su3_stina := fbSu3_stina.bLight;
fbSu3_bra(bOn := eib_su3_bra, bOff := NOT eib_su3_bra, bToggle := fbSu3_2_sw.bLongClick);
su3_bra := fbSu3_bra.bLight;
eib_su3_bra := fbSu3_bra.bLight;
fbSu3_lampa(bOn := eib_su3_lampa, bOff := NOT eib_su3_lampa, bToggle := fbSu3_2_sw.bLongClick);
su3_lampa := fbSu3_lampa.bLight;
su3_kontrazhur := fbSu3_lampa.bLight;
eib_su3_lampa := fbSu3_lampa.bLight;
fbDytjacha(bOn := eib_dytjacha, bOff := NOT eib_dytjacha, bToggle := sw_dytjacha1);
dytjacha := fbDytjacha.bLight;
eib_dytjacha := fbDytjacha.bLight;
fbDytjacha_bra(bOn := eib_dytjacha_bra, bOff := NOT eib_dytjacha_bra, bToggle := sw_dytjacha2);
dytjacha_bra := fbDytjacha_bra.bLight;
eib_dytjacha_bra := fbDytjacha_bra.bLight;
fbGarderob(bOn := eib_garderob, bOff := NOT eib_garderob, bToggle := sw_garderob1);
garderob := fbGarderob.bLight;
eib_garderob := fbGarderob.bLight;
fbServerna(bOn := eib_serverna, bOff := NOT eib_serverna, bToggle := sw_garderob2);
serverna := fbServerna.bLight;
eib_serverna := fbServerna.bLight;
fbKorydor_skeli(duration := lightDuration, sensor := moove_korydor, knx := eib_korydor_skeli);
korydor_skeli := fbKorydor_skeli.out;
eib_korydor_skeli := fbKorydor_skeli.out;
fbKorydor_svitlo(button := sw_korydor, knx := eib_korydor_svitlo);
korydor_svitlo := fbKorydor_svitlo.out;
eib_korydor_svitlo := fbKorydor_svitlo.out;
fbKorydor_lampa(duration := lightDuration, sensor := moove_korydor, knx := eib_korydor_lampa);
korydor_lampa := fbKorydor_lampa.out;
eib_korydor_lampa := fbKorydor_lampa.out;
tambur3_2_long_click_TP(IN := fbTambur3_2_sw.bLongClick, PT := t#500ms);
fbBar(bOn := eib_bar, bOff := NOT eib_bar, bToggle := sw_tambur3_1);
bar := fbBar.bLight;
eib_bar := fbBar.bLight;
fbTambur3_2_sw(bSwitch := sw_tambur3_2, tSwitchTime := longPressDelay);
fbChoven(button := sw_tambur2, duration := lightDuration, sensor := MUX(BOOL_TO_INT(bDarkOutside), TRUE, moove_skhody), knx := eib_choven);
tambur3_2_long_click := tambur3_2_long_click_TP.Q;
choven := fbChoven.out;
eib_choven := fbChoven.out;
fbSpalnya_balkon(bOn := eib_spalnya_balkon, bOff := NOT eib_spalnya_balkon, bToggle := sw_spalnya_balk);
spalnya_balkon := fbSpalnya_balkon.bLight;
eib_spalnya_balkon := fbSpalnya_balkon.bLight;
fbSpalnya_1_sw(bSwitch := sw_spalnya1 XOR sw_spalnya4, tSwitchTime := longPressDelay);
fbSpalnya_light(bOn := eib_spalnya_kulbaba, bOff := NOT eib_spalnya_kulbaba, bToggle := fbSpalnya_1_sw.bShortClick);
spalnya_kulbaba := fbSpalnya_light.bLight;
eib_spalnya_kulbaba := fbSpalnya_light.bLight;
fbShtorySpalnya(bUp := eib_shtory_spalnya_move, bDown := NOT eib_shtory_spalnya_move, bSwitch := fbSpalnya_1_sw.bLongClick, nSetPosition := eib_shtory_spalnya_position, tDriveTime := t#10s, tDriveSwitchOverTime := t#0s, tSwitchOverDeadTime := t#0s);
shtory_open := fbShtorySpalnya.bBlindUp;
shtory_close := fbShtorySpalnya.bBlindDown;
eib_shtory_spalnya_actualPosition := fbShtorySpalnya.nActualPosition;
fbSpalnya_2_sw(bSwitch := sw_spalnya2 XOR sw_spalnya3, tSwitchTime := longPressDelay);
fbSpalnya_kontrazhury(bOn := eib_spalnya_kontrazhury, bOff := NOT eib_spalnya_kontrazhury, bToggle := fbSpalnya_2_sw.bShortClick);
spalnya_kontrazhur := fbSpalnya_kontrazhury.bLight;
spalnya_kontrazhur_b := fbSpalnya_kontrazhury.bLight;
spalnya_kontrazhur_l := fbSpalnya_kontrazhury.bLight;
eib_spalnya_kontrazhury := fbSpalnya_kontrazhury.bLight;
fbTulSpalnya(bUp := eib_tul_spalnya_move, bDown := NOT eib_tul_spalnya_move, bSwitch := fbSpalnya_2_sw.bLongClick, nSetPosition := eib_tul_spalnya_position, tDriveTime := t#10s, tDriveSwitchOverTime := t#0s, tSwitchOverDeadTime := T#0s);
tul_open := fbTulSpalnya.bBlindUp;
tul_close := fbTulSpalnya.bBlindDown;
eib_tul_spalnya_actualPosition := fbTulSpalnya.nActualPosition;
fbSpalnyaLift(bClose := NOT eib_lift_spalnya_move, bOpen := eib_lift_spalnya_move, bSafetyPosition := MAIN.SpalnyaLiftToSafePos, tTurnOffTime := t#20s);
lift_up := fbSpalnyaLift.bWindowOpen;
lift_down := fbSpalnyaLift.bWindowClose;
fbEIB_lift_spalnya_status_SET_RESET(CLAIM := fbSpalnyaLift.bWindowOpen, RELEASE := fbSpalnyaLift.bWindowClose);
eib_lift_spalnya_move := fbEIB_lift_spalnya_status_SET_RESET.BUSY;
tambur3_2_short_click_TP(IN := fbTambur3_2_sw.bShortClick, PT := t#500ms);
tambur3_2_short_click := tambur3_2_short_click_TP.Q;
END_PROGRAM

(* POU lights/fbMoovingSensorLight, ST *)
FUNCTION_BLOCK fbMoovingSensorLight
VAR_INPUT
	button:BOOL;
	duration:TIME;
	sensor:BOOL;
	knx:BOOL;
END_VAR
VAR_OUTPUT
	out: BOOL;
END_VAR
VAR
	fbStairwayLight_00			: FB_StairwellLight;
	button_rising				: R_TRIG;
	sensor_falling				: F_TRIG;
	timer_falling					: F_TRIG;
	knx_falling					: F_TRIG;
	knx_rising					: R_TRIG;
END_VAR

VAR_IN_OUT
END_VAR
knx_rising(CLK:=knx);
knx_falling(CLK:=knx);
button_rising(CLK:=button);
sensor_falling(CLK:= sensor);
timer_falling(clk:=fbStairwayLight_00.bStart);

IF sensor_falling.Q AND NOT out THEN
	fbStairwayLight_00.bOff:=FALSE;
END_IF

fbStairwayLight_00(
	bSwitch:=NOT sensor AND NOT out,
	tLightDuration:=duration,
	tPreWarningStart:=t#100s,
	tPreWarningDuration:=t#500ms);

IF fbStairwayLight_00.bStart THEN
	out := fbStairwayLight_00.bLight;
END_IF

IF timer_falling.Q THEN
	out:=FALSE;
END_IF




IF knx_rising.Q OR knx_falling.Q THEN
	out:= knx;
	IF knx_falling.Q THEN
		fbStairwayLight_00.bOff:=TRUE;
	END_IF
END_IF

IF button_rising.Q THEN
	out:= NOT out;
	fbStairwayLight_00.bOff:=TRUE;
END_IF
END_FUNCTION_BLOCK

(* POU Shtory, CFC *)
PROGRAM Shtory
VAR

END_VAR
VAR (* helpers for the ST form of the networks *)
	_t121 : USINT;
	_t120 : USINT;
END_VAR
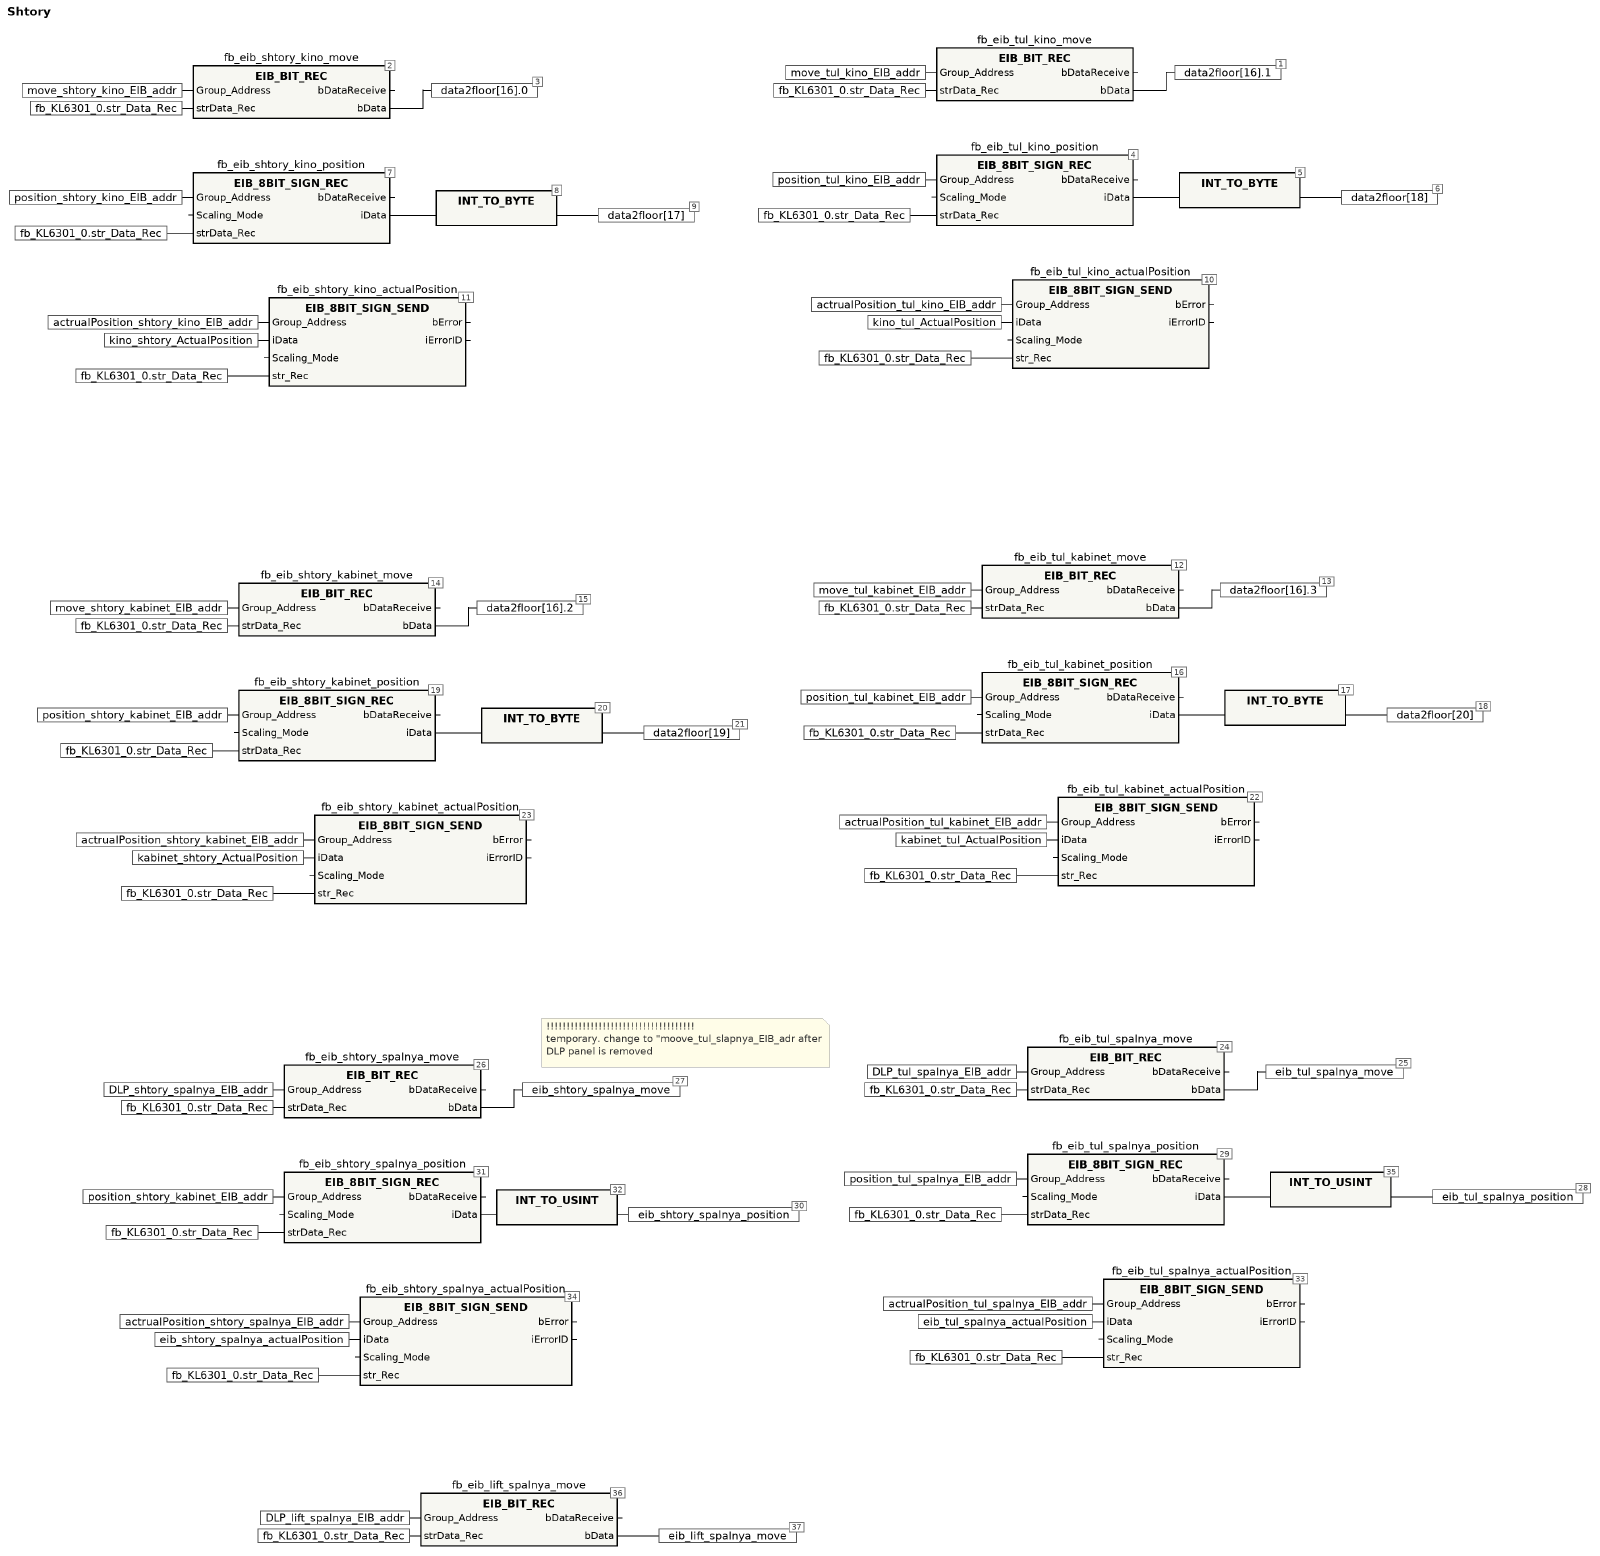
_CFC_ (* Continuous Function Chart, elements in execution order *)
(* !!!!!!!!!!!!!!!!!!!!!!!!!!!!!!!!!!!!! / temporary. change to "moove_tul_slapnya_EIB_adr after DLP panel is removed *)
#0 fb_eib_tul_kino_move:EIB_BIT_REC(Group_Address: move_tul_kino_EIB_addr, strData_Rec: fb_KL6301_0.str_Data_Rec)
#1 data2floor[16].1 <= #0.bData
#2 fb_eib_shtory_kino_move:EIB_BIT_REC(Group_Address: move_shtory_kino_EIB_addr, strData_Rec: fb_KL6301_0.str_Data_Rec)
#3 data2floor[16].0 <= #2.bData
#4 fb_eib_tul_kino_position:EIB_8BIT_SIGN_REC(Group_Address: position_tul_kino_EIB_addr, Scaling_Mode: -, strData_Rec: fb_KL6301_0.str_Data_Rec)
#5 INT_TO_BYTE(#4.iData)
#6 data2floor[18] <= #5
#7 fb_eib_shtory_kino_position:EIB_8BIT_SIGN_REC(Group_Address: position_shtory_kino_EIB_addr, Scaling_Mode: -, strData_Rec: fb_KL6301_0.str_Data_Rec)
#8 INT_TO_BYTE(#7.iData)
#9 data2floor[17] <= #8
#10 fb_eib_tul_kino_actualPosition:EIB_8BIT_SIGN_SEND(Group_Address: actrualPosition_tul_kino_EIB_addr, iData: kino_tul_ActualPosition, Scaling_Mode: -, str_Rec: fb_KL6301_0.str_Data_Rec)
#11 fb_eib_shtory_kino_actualPosition:EIB_8BIT_SIGN_SEND(Group_Address: actrualPosition_shtory_kino_EIB_addr, iData: kino_shtory_ActualPosition, Scaling_Mode: -, str_Rec: fb_KL6301_0.str_Data_Rec)
#12 fb_eib_tul_kabinet_move:EIB_BIT_REC(Group_Address: move_tul_kabinet_EIB_addr, strData_Rec: fb_KL6301_0.str_Data_Rec)
#13 data2floor[16].3 <= #12.bData
#14 fb_eib_shtory_kabinet_move:EIB_BIT_REC(Group_Address: move_shtory_kabinet_EIB_addr, strData_Rec: fb_KL6301_0.str_Data_Rec)
#15 data2floor[16].2 <= #14.bData
#16 fb_eib_tul_kabinet_position:EIB_8BIT_SIGN_REC(Group_Address: position_tul_kabinet_EIB_addr, Scaling_Mode: -, strData_Rec: fb_KL6301_0.str_Data_Rec)
#17 INT_TO_BYTE(#16.iData)
#18 data2floor[20] <= #17
#19 fb_eib_shtory_kabinet_position:EIB_8BIT_SIGN_REC(Group_Address: position_shtory_kabinet_EIB_addr, Scaling_Mode: -, strData_Rec: fb_KL6301_0.str_Data_Rec)
#20 INT_TO_BYTE(#19.iData)
#21 data2floor[19] <= #20
#22 fb_eib_tul_kabinet_actualPosition:EIB_8BIT_SIGN_SEND(Group_Address: actrualPosition_tul_kabinet_EIB_addr, iData: kabinet_tul_ActualPosition, Scaling_Mode: -, str_Rec: fb_KL6301_0.str_Data_Rec)
#23 fb_eib_shtory_kabinet_actualPosition:EIB_8BIT_SIGN_SEND(Group_Address: actrualPosition_shtory_kabinet_EIB_addr, iData: kabinet_shtory_ActualPosition, Scaling_Mode: -, str_Rec: fb_KL6301_0.str_Data_Rec)
#24 fb_eib_tul_spalnya_move:EIB_BIT_REC(Group_Address: DLP_tul_spalnya_EIB_addr, strData_Rec: fb_KL6301_0.str_Data_Rec)
#25 eib_tul_spalnya_move <= #24.bData
#26 fb_eib_shtory_spalnya_move:EIB_BIT_REC(Group_Address: DLP_shtory_spalnya_EIB_addr, strData_Rec: fb_KL6301_0.str_Data_Rec)
#27 eib_shtory_spalnya_move <= #26.bData
#28 eib_tul_spalnya_position <= #35
#29 fb_eib_tul_spalnya_position:EIB_8BIT_SIGN_REC(Group_Address: position_tul_spalnya_EIB_addr, Scaling_Mode: -, strData_Rec: fb_KL6301_0.str_Data_Rec)
#30 eib_shtory_spalnya_position <= #32
#31 fb_eib_shtory_spalnya_position:EIB_8BIT_SIGN_REC(Group_Address: position_shtory_kabinet_EIB_addr, Scaling_Mode: -, strData_Rec: fb_KL6301_0.str_Data_Rec)
#32 INT_TO_USINT(#31.iData)
#33 fb_eib_tul_spalnya_actualPosition:EIB_8BIT_SIGN_SEND(Group_Address: actrualPosition_tul_spalnya_EIB_addr, iData: eib_tul_spalnya_actualPosition, Scaling_Mode: -, str_Rec: fb_KL6301_0.str_Data_Rec)
#34 fb_eib_shtory_spalnya_actualPosition:EIB_8BIT_SIGN_SEND(Group_Address: actrualPosition_shtory_spalnya_EIB_addr, iData: eib_shtory_spalnya_actualPosition, Scaling_Mode: -, str_Rec: fb_KL6301_0.str_Data_Rec)
#35 INT_TO_USINT(#29.iData)
#36 fb_eib_lift_spalnya_move:EIB_BIT_REC(Group_Address: DLP_lift_spalnya_EIB_addr, strData_Rec: fb_KL6301_0.str_Data_Rec)
#37 eib_lift_spalnya_move <= #36.bData
_END_CFC_
(* the same logic as Structured Text *)
(* !!!!!!!!!!!!!!!!!!!!!!!!!!!!!!!!!!!!! / temporary. change to "moove_tul_slapnya_EIB_adr after DLP panel is removed *)
fb_eib_tul_kino_move(Group_Address := move_tul_kino_EIB_addr, strData_Rec := fb_KL6301_0.str_Data_Rec);
data2floor[16].1 := fb_eib_tul_kino_move.bData;
fb_eib_shtory_kino_move(Group_Address := move_shtory_kino_EIB_addr, strData_Rec := fb_KL6301_0.str_Data_Rec);
data2floor[16].0 := fb_eib_shtory_kino_move.bData;
fb_eib_tul_kino_position(Group_Address := position_tul_kino_EIB_addr, strData_Rec := fb_KL6301_0.str_Data_Rec);
data2floor[18] := INT_TO_BYTE(fb_eib_tul_kino_position.iData);
fb_eib_shtory_kino_position(Group_Address := position_shtory_kino_EIB_addr, strData_Rec := fb_KL6301_0.str_Data_Rec);
data2floor[17] := INT_TO_BYTE(fb_eib_shtory_kino_position.iData);
fb_eib_tul_kino_actualPosition(Group_Address := actrualPosition_tul_kino_EIB_addr, iData := kino_tul_ActualPosition, str_Rec := fb_KL6301_0.str_Data_Rec);
fb_eib_shtory_kino_actualPosition(Group_Address := actrualPosition_shtory_kino_EIB_addr, iData := kino_shtory_ActualPosition, str_Rec := fb_KL6301_0.str_Data_Rec);
fb_eib_tul_kabinet_move(Group_Address := move_tul_kabinet_EIB_addr, strData_Rec := fb_KL6301_0.str_Data_Rec);
data2floor[16].3 := fb_eib_tul_kabinet_move.bData;
fb_eib_shtory_kabinet_move(Group_Address := move_shtory_kabinet_EIB_addr, strData_Rec := fb_KL6301_0.str_Data_Rec);
data2floor[16].2 := fb_eib_shtory_kabinet_move.bData;
fb_eib_tul_kabinet_position(Group_Address := position_tul_kabinet_EIB_addr, strData_Rec := fb_KL6301_0.str_Data_Rec);
data2floor[20] := INT_TO_BYTE(fb_eib_tul_kabinet_position.iData);
fb_eib_shtory_kabinet_position(Group_Address := position_shtory_kabinet_EIB_addr, strData_Rec := fb_KL6301_0.str_Data_Rec);
data2floor[19] := INT_TO_BYTE(fb_eib_shtory_kabinet_position.iData);
fb_eib_tul_kabinet_actualPosition(Group_Address := actrualPosition_tul_kabinet_EIB_addr, iData := kabinet_tul_ActualPosition, str_Rec := fb_KL6301_0.str_Data_Rec);
fb_eib_shtory_kabinet_actualPosition(Group_Address := actrualPosition_shtory_kabinet_EIB_addr, iData := kabinet_shtory_ActualPosition, str_Rec := fb_KL6301_0.str_Data_Rec);
fb_eib_tul_spalnya_move(Group_Address := DLP_tul_spalnya_EIB_addr, strData_Rec := fb_KL6301_0.str_Data_Rec);
eib_tul_spalnya_move := fb_eib_tul_spalnya_move.bData;
fb_eib_shtory_spalnya_move(Group_Address := DLP_shtory_spalnya_EIB_addr, strData_Rec := fb_KL6301_0.str_Data_Rec);
eib_shtory_spalnya_move := fb_eib_shtory_spalnya_move.bData;
eib_tul_spalnya_position := _t121;
fb_eib_tul_spalnya_position(Group_Address := position_tul_spalnya_EIB_addr, strData_Rec := fb_KL6301_0.str_Data_Rec);
eib_shtory_spalnya_position := _t120;
fb_eib_shtory_spalnya_position(Group_Address := position_shtory_kabinet_EIB_addr, strData_Rec := fb_KL6301_0.str_Data_Rec);
_t120 := INT_TO_USINT(fb_eib_shtory_spalnya_position.iData);
fb_eib_tul_spalnya_actualPosition(Group_Address := actrualPosition_tul_spalnya_EIB_addr, iData := eib_tul_spalnya_actualPosition, str_Rec := fb_KL6301_0.str_Data_Rec);
fb_eib_shtory_spalnya_actualPosition(Group_Address := actrualPosition_shtory_spalnya_EIB_addr, iData := eib_shtory_spalnya_actualPosition, str_Rec := fb_KL6301_0.str_Data_Rec);
_t121 := INT_TO_USINT(fb_eib_tul_spalnya_position.iData);
fb_eib_lift_spalnya_move(Group_Address := DLP_lift_spalnya_EIB_addr, strData_Rec := fb_KL6301_0.str_Data_Rec);
eib_lift_spalnya_move := fb_eib_lift_spalnya_move.bData;
END_PROGRAM

(* POU HVAC/seasonChange, ST *)
PROGRAM seasonChange
VAR
	OATfilter						: FB_PT2;
	OAT_FILTER_T1				: TIME := t#5s;
	OAT_FILTER_T2				: TIME := t#4h;
END_VAR
OATfilter.bSetActual := MAIN.init;

IF NOT EIB.fb_heating_setpoint_read.bDataReceive THEN
	heatingOnOATSp := REAL_TO_INT (EIB.fb_heating_setpoint_read.rData);
END_IF;

IF NOT EIB.fb_cooling_setpoint_read.bDataReceive THEN
	coolingOnOATSp := REAL_TO_INT (EIB.fb_cooling_setpoint_read.rData);
END_IF;

IF NOT EIB.fb_climateControlMode_read.bDataReceive THEN
	climateControlMode := BYTE_TO_INT(EIB.eib_byte_climate_control_mode);
END_IF;


OATfilter(fIn := OAT, tT1 := OAT_FILTER_T1, tT2 := OAT_FILTER_T2, fOut => filteredOAT);
IF climateControlMode = 0 THEN

	IF filteredOAT > coolingOnOATSp THEN
		RTControlMode 		:= 2;
	END_IF;

	IF filteredOAT < heatingOnOATSp THEN
		RTControlMode 		:= 1;
	END_IF;
ELSE
	IF climateControlMode = 1 THEN
		RTControlMode		:= 1;
	END_IF;

	IF climateControlMode = 3 THEN
		RTControlMode		:= 2;
	END_IF;

	IF climateControlMode = 9 THEN
		RTControlMode		:= 0;
	END_IF;

END_IF;

CASE RTControlMode OF
	Off:
		heatingPumpOn 		:= FALSE;
		freeCoolingValveOn	:= FALSE;
	Heating:
		heatingPumpOn		:= TRUE;
		freeCoolingValveOn	:= FALSE;
	Cooling:
		heatingPumpOn		:= TRUE;
		freeCoolingValveOn	:= TRUE;
END_CASE;
END_PROGRAM

(* POU HVAC/climate, ST *)
PROGRAM climate
VAR
	t_tambur: REAL;
	t_su: REAL;
	t_spalnya: REAL;
(*
	t_max: REAL;
	t_min: REAL;
*)
	OAT_filter: 						FB_PT1;
	t_tambur_filter: 					FB_PT1;
	t_su_filter: 						FB_PT1;
	t_spalnya_filter: 					FB_PT1;
	fb_freshbarFloorHeating: 			fbPWM;
	fb_garderobFloorHeating: 		fbPWM;
	fb_spalnyaFloorHeating: 			fbPWM;
	fb_servernaFloorHeating: 		fbPWM;
	fb_su3FloorHeating: 				fbPWM;
	fb_dytjachaFloorHeating: 		fbPWM;

	temperatureFiltersCycleTime: 		TIME := t#28ms;
	temperaturesFilterT1: 			TIME := t#12m;
	temp: REAL;
END_VAR
(*фільтри показань сенсорів температури*)
OAT_filter.bSetActual := MAIN.init;
OAT_filter.tCycletime:=temperatureFiltersCycleTime;
OAT_filter.tT1:=temperaturesFilterT1;
OAT_filter(fIn:=INT_TO_REAL(iT_out)/10);
t_out := TRUNC(OAT_filter.fOut*100)/100.0;
OAT:=REAL_TO_INT(t_out);



floorHeating;
(*

IF VITALNYA_HVAC.heat_mode=0 THEN
				VITALNYA_HVAC.fancoil_speed:=0;
				(*VITALNYA_HVAC.collector:=2#00000000; all closed*)
				VITALNYA_HVAC.klapan:=16#7FFF;(*full closed*)
				VITALNYA_HVAC.zaslinka:=TRUE;(*closed*)
	END_IF

	IF KINO_HVAC.heat_mode=0 THEN
				KINO_HVAC.fancoil_speed:=0;
				(*KINO_HVAC.collector:=2#00000000; all closed*)
				KINO_HVAC.klapan:=16#7FFF;(*full closed*)
				KINO_HVAC.zaslinka:=TRUE;(*closed*)
	END_IF

	IF STUDIO_HVAC.heat_mode=0 THEN
				STUDIO_HVAC.fancoil_speed:=0;
				(*STUDIO_HVAC.collector:=2#00000000; all closed*)
				STUDIO_HVAC.klapan:=16#7FFF;(*full closed*)
				STUDIO_HVAC.zaslinka:=TRUE;(*closed*)
	END_IF

	IF KABINET_HVAC.heat_mode=0 THEN
				KABINET_HVAC.fancoil_speed:=0;
				(*KABINET_HVAC.collector:=2#00000000; all closed*)
				KABINET_HVAC.klapan:=16#7FFF;(*full closed*)
				KABINET_HVAC.zaslinka:=TRUE;(*closed*)
	END_IF

	IF DYTJACHA_HVAC.heat_mode=0 THEN
				DYTJACHA_HVAC.fancoil_speed:=0;
				(*DYTJACHA_HVAC.collector:=2#00000000; all closed*)
				DYTJACHA_HVAC.klapan:=16#7FFF;(*full closed*)
				DYTJACHA_HVAC.zaslinka:=TRUE;(*closed*)
	END_IF

	IF SPALNYA_HVAC.heat_mode=0 THEN
				SPALNYA_HVAC.fancoil_speed:=0;
				(*SPALNYA_HVAC.collector:=2#00000000; all closed*)
				SPALNYA_HVAC.klapan:=16#7FFF;(*full closed*)
				SPALNYA_HVAC.zaslinka:=TRUE;(*closed*)
	END_IF
*)





(*локальні змінні для фенкойлів 3го поверхну об'явлені в області виходів*)

(*------------------------fancoil speed --------------------------------------------------*)
IF EIB.fb_vitalnya_damper_ctrl_rec.bData THEN
	vitalnya_hvac.fancoil_speed:=3;
ELSE
	IF vitalnya_HVAC.heating_signal = 0  THEN
		CASE vitalnya_hvac.fancoil_speed OF
			0:	IF vitalnya_hvac.cooling_signal>0 THEN vitalnya_HVAC.fancoil_speed:=1; END_IF

			1:	IF vitalnya_hvac.cooling_signal=0 THEN vitalnya_HVAC.fancoil_speed:=0; END_IF
				IF vitalnya_hvac.cooling_signal>50 THEN  vitalnya_HVAC.fancoil_speed:=2; END_IF

			2:	IF vitalnya_hvac.cooling_signal=0 THEN vitalnya_HVAC.fancoil_speed:=0; END_IF
				IF vitalnya_hvac.cooling_signal>75  THEN vitalnya_HVAC.fancoil_speed:=3; END_IF
				IF vitalnya_hvac.cooling_signal<25  THEN vitalnya_HVAC.fancoil_speed:=1; END_IF

			3:	IF vitalnya_hvac.cooling_signal=0 THEN vitalnya_HVAC.fancoil_speed:=0; END_IF
				IF vitalnya_hvac.cooling_signal<50  THEN vitalnya_HVAC.fancoil_speed:=2; END_IF
		END_CASE
	END_IF

	IF vitalnya_HVAC.cooling_signal = 0 THEN
		CASE vitalnya_hvac.fancoil_speed OF
			0:	IF vitalnya_hvac.heating_signal>0 THEN vitalnya_HVAC.fancoil_speed:=1; END_IF

			1:	IF vitalnya_hvac.heating_signal=0 THEN vitalnya_HVAC.fancoil_speed:=0; END_IF
				IF vitalnya_hvac.heating_signal>50 THEN  vitalnya_HVAC.fancoil_speed:=2; END_IF

			2:	IF vitalnya_hvac.heating_signal=0 THEN vitalnya_HVAC.fancoil_speed:=0; END_IF
				IF vitalnya_hvac.heating_signal>75  THEN vitalnya_HVAC.fancoil_speed:=3; END_IF
				IF vitalnya_hvac.heating_signal<25  THEN vitalnya_HVAC.fancoil_speed:=1; END_IF

			3:	IF vitalnya_hvac.heating_signal=0 THEN vitalnya_HVAC.fancoil_speed:=0; END_IF
				IF vitalnya_hvac.heating_signal<50  THEN vitalnya_HVAC.fancoil_speed:=2; END_IF
		END_CASE
	END_IF
END_IF

IF EIB.fb_kino_damper_ctrl_rec.bData THEN
	kino_hvac.fancoil_speed:=3;
ELSE
	IF kino_HVAC.heating_signal = 0 THEN
		CASE kino_hvac.fancoil_speed OF
			0:	IF kino_hvac.cooling_signal>0 THEN kino_HVAC.fancoil_speed:=1; END_IF

			1:	IF kino_hvac.cooling_signal=0 THEN kino_HVAC.fancoil_speed:=0; END_IF
				IF kino_hvac.cooling_signal>50 THEN  kino_HVAC.fancoil_speed:=2; END_IF

			2:	IF kino_hvac.cooling_signal=0 THEN kino_HVAC.fancoil_speed:=0; END_IF
				IF kino_hvac.cooling_signal>75  THEN kino_HVAC.fancoil_speed:=3; END_IF
				IF kino_hvac.cooling_signal<25  THEN kino_HVAC.fancoil_speed:=1; END_IF

			3:	IF kino_hvac.cooling_signal=0 THEN kino_HVAC.fancoil_speed:=0; END_IF
				IF kino_hvac.cooling_signal<50  THEN kino_HVAC.fancoil_speed:=2; END_IF
		END_CASE
	END_IF
	IF kino_HVAC.cooling_signal = 0 THEN
		CASE kino_hvac.fancoil_speed OF
			0:	IF kino_hvac.heating_signal>0 THEN kino_HVAC.fancoil_speed:=1; END_IF

			1:	IF kino_hvac.heating_signal=0 THEN kino_HVAC.fancoil_speed:=0; END_IF
				IF kino_hvac.heating_signal>50 THEN  kino_HVAC.fancoil_speed:=2; END_IF

			2:	IF kino_hvac.heating_signal=0 THEN kino_HVAC.fancoil_speed:=0; END_IF
				IF kino_hvac.heating_signal>75  THEN kino_HVAC.fancoil_speed:=3; END_IF
				IF kino_hvac.heating_signal<25  THEN kino_HVAC.fancoil_speed:=1; END_IF

			3:	IF kino_hvac.heating_signal=0 THEN kino_HVAC.fancoil_speed:=0; END_IF
				IF kino_hvac.heating_signal<50  THEN kino_HVAC.fancoil_speed:=2; END_IF
		END_CASE
	END_IF
END_IF

IF EIB.fb_kabinet_damper_ctrl_rec.bData THEN
	kabinet_hvac.fancoil_speed:=3;
ELSE
	IF kabinet_HVAC.heating_signal = 0 THEN
		CASE kabinet_hvac.fancoil_speed OF
			0:	IF kabinet_hvac.cooling_signal>0 THEN kabinet_HVAC.fancoil_speed:=1; END_IF

			1:	IF kabinet_hvac.cooling_signal=0 THEN kabinet_HVAC.fancoil_speed:=0; END_IF
				IF kabinet_hvac.cooling_signal>50 THEN  kabinet_HVAC.fancoil_speed:=2; END_IF

			2:	IF kabinet_hvac.cooling_signal=0 THEN kabinet_HVAC.fancoil_speed:=0; END_IF
				IF kabinet_hvac.cooling_signal>75  THEN kabinet_HVAC.fancoil_speed:=3; END_IF
				IF kabinet_hvac.cooling_signal<25  THEN kabinet_HVAC.fancoil_speed:=1; END_IF

			3:	IF kabinet_hvac.cooling_signal=0 THEN kabinet_HVAC.fancoil_speed:=0; END_IF
				IF kabinet_hvac.cooling_signal<50  THEN kabinet_HVAC.fancoil_speed:=2; END_IF
		END_CASE
	END_IF
	IF kabinet_HVAC.cooling_signal = 0 THEN
		CASE kabinet_hvac.fancoil_speed OF
			0:	IF kabinet_hvac.heating_signal>0 THEN kabinet_HVAC.fancoil_speed:=1; END_IF

			1:	IF kabinet_hvac.heating_signal=0 THEN kabinet_HVAC.fancoil_speed:=0; END_IF
				IF kabinet_hvac.heating_signal>50 THEN  kabinet_HVAC.fancoil_speed:=2; END_IF

			2:	IF kabinet_hvac.heating_signal=0 THEN kabinet_HVAC.fancoil_speed:=0; END_IF
				IF kabinet_hvac.heating_signal>75  THEN kabinet_HVAC.fancoil_speed:=3; END_IF
				IF kabinet_hvac.heating_signal<25  THEN kabinet_HVAC.fancoil_speed:=1; END_IF

			3:	IF kabinet_hvac.heating_signal=0 THEN kabinet_HVAC.fancoil_speed:=0; END_IF
				IF kabinet_hvac.heating_signal<50  THEN kabinet_HVAC.fancoil_speed:=2; END_IF
		END_CASE
	END_IF
END_IF

IF EIB.fb_dytjacha_damper_ctrl_rec.bData THEN
	dytjacha_hvac.fancoil_speed:=3;
ELSE
	IF dytjacha_HVAC.heating_signal = 0 THEN
		CASE dytjacha_hvac.fancoil_speed OF
			0:	IF dytjacha_hvac.cooling_signal>0 THEN dytjacha_HVAC.fancoil_speed:=1; END_IF

			1:	IF dytjacha_hvac.cooling_signal=0 THEN dytjacha_HVAC.fancoil_speed:=0; END_IF
				IF dytjacha_hvac.cooling_signal>50 THEN  dytjacha_HVAC.fancoil_speed:=2; END_IF

			2:	IF dytjacha_hvac.cooling_signal=0 THEN dytjacha_HVAC.fancoil_speed:=0; END_IF
				IF dytjacha_hvac.cooling_signal>75  THEN dytjacha_HVAC.fancoil_speed:=3; END_IF
				IF dytjacha_hvac.cooling_signal<25  THEN dytjacha_HVAC.fancoil_speed:=1; END_IF

			3:	IF dytjacha_hvac.cooling_signal=0 THEN dytjacha_HVAC.fancoil_speed:=0; END_IF
				IF dytjacha_hvac.cooling_signal<50  THEN dytjacha_HVAC.fancoil_speed:=2; END_IF
		END_CASE
	END_IF
	IF dytjacha_HVAC.cooling_signal = 0 THEN
		CASE dytjacha_hvac.fancoil_speed OF
			0:	IF dytjacha_hvac.heating_signal>0 THEN dytjacha_HVAC.fancoil_speed:=1; END_IF

			1:	IF dytjacha_hvac.heating_signal=0 THEN dytjacha_HVAC.fancoil_speed:=0; END_IF
				IF dytjacha_hvac.heating_signal>50 THEN  dytjacha_HVAC.fancoil_speed:=2; END_IF

			2:	IF dytjacha_hvac.heating_signal=0 THEN dytjacha_HVAC.fancoil_speed:=0; END_IF
				IF dytjacha_hvac.heating_signal>75  THEN dytjacha_HVAC.fancoil_speed:=3; END_IF
				IF dytjacha_hvac.heating_signal<25  THEN dytjacha_HVAC.fancoil_speed:=1; END_IF

			3:	IF dytjacha_hvac.heating_signal=0 THEN dytjacha_HVAC.fancoil_speed:=0; END_IF
				IF dytjacha_hvac.heating_signal<50  THEN dytjacha_HVAC.fancoil_speed:=2; END_IF
		END_CASE
	END_IF
END_IF

IF EIB.fb_spalnya_damper_ctrl_rec.bData THEN
	spalnya_hvac.fancoil_speed:=3;
ELSE
	IF spalnya_HVAC.heating_signal = 0 THEN
		CASE spalnya_hvac.fancoil_speed OF
			0:	IF spalnya_hvac.cooling_signal>0 THEN spalnya_HVAC.fancoil_speed:=1; END_IF

			1:	IF spalnya_hvac.cooling_signal=0 THEN spalnya_HVAC.fancoil_speed:=0; END_IF
				IF spalnya_hvac.cooling_signal>50 THEN  spalnya_HVAC.fancoil_speed:=2; END_IF

			2:	IF spalnya_hvac.cooling_signal=0 THEN spalnya_HVAC.fancoil_speed:=0; END_IF
				IF spalnya_hvac.cooling_signal>75  THEN spalnya_HVAC.fancoil_speed:=3; END_IF
				IF spalnya_hvac.cooling_signal<25  THEN spalnya_HVAC.fancoil_speed:=1; END_IF

			3:	IF spalnya_hvac.cooling_signal=0 THEN spalnya_HVAC.fancoil_speed:=0; END_IF
				IF spalnya_hvac.cooling_signal<50  THEN spalnya_HVAC.fancoil_speed:=2; END_IF
		END_CASE
	END_IF
	IF spalnya_HVAC.cooling_signal = 0 THEN
		CASE spalnya_hvac.fancoil_speed OF
			0:	IF spalnya_hvac.heating_signal>0 THEN spalnya_HVAC.fancoil_speed:=1; END_IF

			1:	IF spalnya_hvac.heating_signal=0 THEN spalnya_HVAC.fancoil_speed:=0; END_IF
				IF spalnya_hvac.heating_signal>50 THEN  spalnya_HVAC.fancoil_speed:=2; END_IF

			2:	IF spalnya_hvac.heating_signal=0 THEN spalnya_HVAC.fancoil_speed:=0; END_IF
				IF spalnya_hvac.heating_signal>75  THEN spalnya_HVAC.fancoil_speed:=3; END_IF
				IF spalnya_hvac.heating_signal<25  THEN spalnya_HVAC.fancoil_speed:=1; END_IF

			3:	IF spalnya_hvac.heating_signal=0 THEN spalnya_HVAC.fancoil_speed:=0; END_IF
				IF spalnya_hvac.heating_signal<50  THEN spalnya_HVAC.fancoil_speed:=2; END_IF
		END_CASE
	END_IF
END_IF
CASE DYTJACHA_HVAC.fancoil_speed OF
	0:	fancoil_dytjacha_low:=FALSE;
		fancoil_dytjacha_med:=FALSE;
		fancoil_dytjacha_high:=FALSE;

	1:	fancoil_dytjacha_low:=TRUE;
		fancoil_dytjacha_med:=FALSE;
		fancoil_dytjacha_high:=FALSE;

	2:	fancoil_dytjacha_low:=FALSE;
		fancoil_dytjacha_med:=TRUE;
		fancoil_dytjacha_high:=FALSE;

	3:	fancoil_dytjacha_low:=FALSE;
		fancoil_dytjacha_med:=FALSE;
		fancoil_dytjacha_high:=TRUE;
END_CASE

CASE SPALNYA_HVAC.fancoil_speed OF
	0:	fancoil_spalnya_low:=FALSE;
		fancoil_spalnya_med:=FALSE;
		fancoil_spalnya_high:=FALSE;

	1:	fancoil_spalnya_low:=TRUE;
		fancoil_spalnya_med:=FALSE;
		fancoil_spalnya_high:=FALSE;

	2:	fancoil_spalnya_low:=FALSE;
		fancoil_spalnya_med:=TRUE;
		fancoil_spalnya_high:=FALSE;

	3:	fancoil_spalnya_low:=FALSE;
		fancoil_spalnya_med:=TRUE; (*ПОМЕНЯТЬ ОБРАТНО ЗАМЕНИЛ ИЗ-ЗА НЕРАБОТАЮЩЕЙ 3й  СКОРОСТИ  ФАНКОЙЛА 17-10-2016*)
		fancoil_spalnya_high:=FALSE;
END_CASE
CASE KABINET_HVAC.fancoil_speed OF
	0:	data2floor[0].0:=0; (*запис в масив даних, що відправляються на 2й поверх*)
		data2floor[0].1:=0;
		data2floor[0].2:=0;

	1:	data2floor[0].0:=1; (*запис в масив даних, що відправляються на 2й поверх*)
		data2floor[0].1:=0;
		data2floor[0].2:=0;

	2:	data2floor[0].0:=0; (*запис в масив даних, що відправляються на 2й поверх*)
		data2floor[0].1:=1;
		data2floor[0].2:=0;

	3:	data2floor[0].0:=0; (*запис в масив даних, що відправляються на 2й поверх*)
		data2floor[0].1:=0;
		data2floor[0].2:=1;
END_CASE

CASE KINO_HVAC.fancoil_speed OF
	0:	data2floor[0].3:=0; (*запис в масив даних, що відправляються на 2й поверх*)
		data2floor[0].4:=0;
		data2floor[0].5:=0;

	1:	data2floor[0].3:=1; (*запис в масив даних, що відправляються на 2й поверх*)
		data2floor[0].4:=0;
		data2floor[0].5:=0;

	2:	data2floor[0].3:=0; (*запис в масив даних, що відправляються на 2й поверх*)
		data2floor[0].4:=1;
		data2floor[0].5:=0;

	3:	data2floor[0].3:=0; (*запис в масив даних, що відправляються на 2й поверх*)
		data2floor[0].4:=0;
		data2floor[0].5:=1;
END_CASE

CASE VITALNYA_HVAC.fancoil_speed OF
	0:	data1floor[0].0:=0; (*запис в масив даних, що відправляються на 1й поверх*)
		data1floor[0].1:=0;
		data1floor[0].2:=0;

	1:	data1floor[0].0:=1; (*запис в масив даних, що відправляються на 1й поверх*)
		data1floor[0].1:=0;
		data1floor[0].2:=0;

	2:	data1floor[0].0:=0; (*запис в масив даних, що відправляються на 1й поверх*)
		data1floor[0].1:=1;
		data1floor[0].2:=0;

	3:	data1floor[0].0:=0; (*запис в масив даних, що відправляються на 1й поверх*)
		data1floor[0].1:=0;
		data1floor[0].2:=1;
END_CASE

(*--------------------------------------klapany--------------------------------------------*)
(*data1floor[2]:=WORD_TO_BYTE(VITALNYA_HVAC.klapan); data1floor[3]:=WORD_TO_BYTE(SHR(VITALNYA_HVAC.klapan,8));*)
klapan_vitalnya:=VITALNYA_HVAC.klapan;
klapan_spalnya:=SPALNYA_HVAC.klapan;
klapan_dytjacha:=DYTJACHA_HVAC.klapan;

data2floor[2]:=WORD_TO_BYTE(KABINET_HVAC.klapan); data2floor[3]:=WORD_TO_BYTE(SHR(KABINET_HVAC.klapan,8));
data2floor[4]:=WORD_TO_BYTE(KINO_HVAC.klapan); data2floor[5]:=WORD_TO_BYTE(SHR(KINO_HVAC.klapan,8));

(*------------------------------zaslinky------------------------------------*)
z_vitalnya:=VITALNYA_HVAC.zaslinka;
z_kabinet:=KABINET_HVAC.zaslinka;
z_kino:=KINO_HVAC.zaslinka;
z_dytjacha:=DYTJACHA_HVAC.zaslinka;
z_spalnya:=SPALNYA_HVAC.zaslinka;

(*-----------------------------tepla pidloga-------------------------------*)
data1floor[0].4:=VITALNYA_HVAC.floor_heating;
data2floor[1].0:=KABINET_HVAC.floor_heating;
data2floor[1].1:=KABINET_HVAC.floor_heating;
data2floor[1].2:=STUDIO_HVAC.floor_heating;
data2floor[1].3:=STUDIO_HVAC.floor_heating;
END_PROGRAM
ACTION floorHeating:
t_tambur_filter.tCycletime:=temperatureFiltersCycleTime;
t_tambur_filter.tT1:=temperaturesFilterT1;
t_tambur_filter (fIn:=INT_TO_REAL(iT_tambur)/10, fOut=>t_tambur);

t_su_filter.tCycletime:=temperatureFiltersCycleTime;
t_su_filter.tT1:=temperaturesFilterT1;
t_su_filter(fIn:=INT_TO_REAL(iT_su)/10, fOut=>t_su);

t_spalnya_filter.tCycletime:=temperatureFiltersCycleTime;
t_spalnya_filter.tT1:=temperaturesFilterT1;
t_spalnya_filter(fIn:=INT_TO_REAL(iT_spalnya)/10, fOut=>t_spalnya);


fb_freshbarFloorHeating(enable := TRUE, cycleLength:= t#10m, pulseWidth := freshbarFloorHeatingSp);
freshbar_col := fb_freshbarFloorHeating.out;

fb_servernaFloorHeating(enable := TRUE, cycleLength:= t#10m, pulseWidth := servernaFloorHeatingSp);
serverna_col := fb_servernaFloorHeating.out;
korydor_col := fb_servernaFloorHeating.out;

fb_su3FloorHeating(enable := TRUE, cycleLength:= t#10m, pulseWidth := su3FloorHeatingSp);
su_col_pidloga := fb_su3FloorHeating.out;
su_col_stina := fb_su3FloorHeating.out;

fb_spalnyaFloorHeating(enable := TRUE, cycleLength:= t#10m, pulseWidth := spalnyaFloorHeatingSp);
spalnya_col := fb_spalnyaFloorHeating.out;

fb_dytjachaFloorHeating (enable := TRUE, cycleLength:= t#10m, pulseWidth := dytjachaFloorHeatingSp);
dytjacha_col := fb_dytjachaFloorHeating.out;
(*
t_max:=70;
t_min:=20;
IF t_out<15 THEN

	IF t_tambur > t_max THEN (*вимкнути колектор, якщо підлога тепліша за верхню межу температури*)
		freshbar_col:=FALSE;
	ELSE
		IF t_tambur< t_min THEN (*увімкнути колектор, якщо підлога холодніша за нижню межу*)
			freshbar_col:=TRUE;
		ELSE
			freshbar_col:= FALSE; (*ПОСТАВИТИ В ЗАЛЕЖНІСТЬ ВІД ЗОВНІШНЬОЇ ТЕМПЕРАТУРИ*)
		END_IF
	END_IF

	IF t_su > t_max THEN
		su_col_pidloga:=FALSE;
		su_col_stina:=FALSE;
			serverna_col:=FALSE;
	ELSE
		IF t_su< t_min THEN
			su_col_pidloga:=TRUE;
			su_col_stina:=TRUE;
			serverna_col:=TRUE;
		ELSE
			su_col_pidloga:=FALSE; (*ПОСТАВИТИ В ЗАЛЕЖНІСТЬ ВІД ЗОВНІШНЬОЇ ТЕМПЕРАТУРИ*)
			su_col_stina:=FALSE;
			serverna_col:=FALSE;
		END_IF
	END_IF

	IF t_spalnya>t_max THEN (*щоб не вистигала підлога*)
		spalnya_col:=FALSE;
	ELSE
		IF t_spalnya<t_min THEN
			spalnya_col:=TRUE;
		ELSE
			spalnya_col:=SPALNYA_HVAC.floor_heating;
		END_IF
	END_IF


END_IF
*)
END_ACTION

(* POU fbPWM, ST *)
FUNCTION_BLOCK fbPWM
VAR_INPUT
	enable				: BOOL 		:= TRUE;
	cycleLength			: TIME 		:= t#10m;
	pulseWidth			: INT		:= 100; (*0-100%*)
END_VAR
VAR_OUTPUT
	out					: BOOL;
END_VAR
VAR
	pulseTimer			: TP;
	gapTimer			: TP;
	pulseLength			: TIME;
	temp				: REAL;
END_VAR
temp:= TIME_TO_REAL(cycleLength) * (INT_TO_REAL(pulseWidth)/100);
pulseLength := REAL_TO_TIME(temp );
gapTimer(IN := enable AND NOT pulseTimer.Q, PT := cycleLength-pulseLength);
pulseTimer(IN := enable AND NOT gapTimer.Q, PT := pulseLength, q=>out);
END_FUNCTION_BLOCK

(* POU ADS_write, ST *)
PROGRAM ADS_write
VAR
	write_timeout: TIME;
	b_write1, b_write2: BOOL;
	write_ads1, write_ads2, write_ads4: ADSWRITE;

	timer1, timer2:TP;
	errorcounter1, errorcounter2, pack_c:CTU ;
	test_word: WORD;
	i2,j2,i1,j1, i4,j4: INT;
	data_changed: BOOL;
	try_again2, try_again1, try_again4: BOOL;
	timer4: TP;
	b_write4: BOOL;
	errorcounter4: CTU;
END_VAR
write_timeout:=t#3s;

timer2(PT:=write_timeout*2);
timer2.IN:=FALSE;



FOR 2i:=0 TO (SIZEOF(data2floor))-1 DO
	IF data2floor[i2]<>data2floor_prev[i2]  OR try_again2 THEN
		b_write2:=TRUE;
		EXIT;
	ELSE
		b_write2:=FALSE;
	END_IF
END_FOR


FOR i1:=0 TO (SIZEOF(data1floor))-1 DO
	IF data1floor[i1]<>data1floor_prev[i1]  OR try_again1 THEN
		b_write1:=TRUE;
		EXIT;
	ELSE
		b_write1:=FALSE;
	END_IF
END_FOR


FOR i4:=0 TO (SIZEOF(data_derevo))-1 DO
	IF data_derevo[i4]<>data_derevo[i4]  OR try_again4 THEN
		b_write4:=TRUE;
		EXIT;
	ELSE
		b_write4:=FALSE;
	END_IF
END_FOR



(*
IF write_ads2.BUSY THEN b_write2:=FALSE; END_IF

	write_ads2(
		NETID:=ads_adr2,
		PORT:=800,
		IDXGRP:=16#4020,
		IDXOFFS:=300,
		WRITE:=b_write2,
		TMOUT:=write_timeout,
		LEN:=SIZEOF(data2floor),
		SRCADDR:=ADR(data2floor));
write_ads2.WRITE:=FALSE;

IF write_ads2.ERR AND NOT timer2.Q THEN
	timer2.IN:=TRUE;
	try_again2:=TRUE;
ELSE try_again2:=FALSE;
END_IF


(*1floor*)
FOR i1:=0 TO (SIZEOF(data1floor))-1 DO
	IF data1floor[i1]<>data1floor_prev[i1] AND NOT timer1.Q THEN
		b_write1:=TRUE;
		EXIT;
	ELSE
		b_write1:=FALSE;
	END_IF
END_FOR

IF try_again1 AND NOT timer1.Q THEN
	b_write1:=TRUE;
	try_again1:=FALSE;
END_IF

errorcounter1(cu:=write_ads1.ERR);

IF write_ads1.BUSY THEN b_write1:=FALSE; END_IF

	write_ads1(
		NETID:=ads_adr1,
		PORT:=800,
		IDXGRP:=16#4020,
		IDXOFFS:=300,
		WRITE:=b_write1,
		TMOUT:=write_timeout,
		LEN:=SIZEOF(data1floor),
		SRCADDR:=ADR(data1floor));

IF write_ads1.ERR AND NOT timer1.Q THEN
	timer1.IN:=TRUE;
	try_again1:=TRUE;
END_IF
timer1(PT:=write_timeout);
timer1.IN:=FALSE;



(*derevo*)
FOR i4:=0 TO (SIZEOF(data_derevo))-1 DO
	IF data_derevo[i4]<>data_derevo_prev[i4] AND NOT timer4.Q THEN
		b_write4:=TRUE;
		EXIT;
	ELSE
		b_write4:=FALSE;
	END_IF
END_FOR

IF try_again4 AND NOT timer4.Q THEN
	b_write4:=TRUE;
	try_again4:=FALSE;
END_IF

errorcounter4(cu:=write_ads4.ERR);


IF write_ads4.BUSY THEN b_write4:=FALSE; END_IF

	write_ads4(
		NETID:=ads_adr4,
		PORT:=800,
		IDXGRP:=16#4020,
		IDXOFFS:=400,
		WRITE:=b_write4,
		TMOUT:=write_timeout,
		LEN:=SIZEOF(data_derevo),
		SRCADDR:=ADR(data_derevo));

IF write_ads4.ERR AND NOT timer4.Q THEN
	timer4.IN:=TRUE;
	try_again4:=TRUE;
END_IF
timer4(PT:=write_timeout);
timer4.IN:=FALSE;
*)

FOR j1:=0 TO (SIZEOF(data1floor))-1 DO
	data1floor_prev[j1]:=data1floor[j1];
END_FOR

FOR j:=0 TO (SIZEOF(data2floor))-1 DO
	data2floor_prev[j]:=data2floor[j];
END_FOR

FOR j4:=0 TO (SIZEOF(data_derevo))-1 DO
	data_derevo_prev[j4]:=data_derevo[j4];
END_FOR
END_PROGRAM

(* POU ADS_Communication, CFC *)
PROGRAM ADS_Communication
VAR

	fb_floor1ADSwrite: ADSWRITE;
	fb_floor2ADSwrite: ADSWRITE;
	fb_floor4ADSwrite: ADSWRITE;
	fb_gymADSwrite: ADSWRITE;

	heartbeat:TP;
	timeout : TIME := t#2s;

END_VAR
VAR (* helpers for the ST form of the networks *)
	_t99 : BOOL;
	_t96 : BOOL;
END_VAR
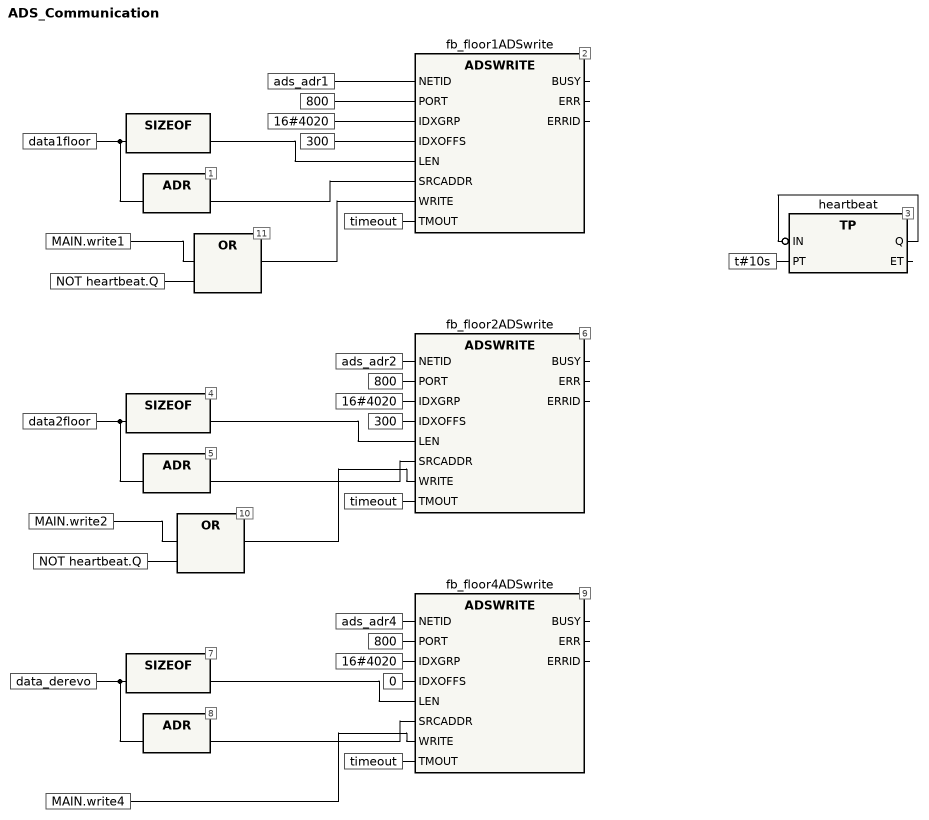
_CFC_ (* Continuous Function Chart, elements in execution order *)
#0 SIZEOF(data1floor)
#1 ADR(data1floor)
#2 fb_floor1ADSwrite:ADSWRITE(NETID: ads_adr1, PORT: 800, IDXGRP: 16#4020, IDXOFFS: 300, LEN: #0, SRCADDR: #1, WRITE: #11, TMOUT: timeout)
#3 heartbeat:TP(IN: NOT #3.Q, PT: t#10s)
#4 SIZEOF(data2floor)
#5 ADR(data2floor)
#6 fb_floor2ADSwrite:ADSWRITE(NETID: ads_adr2, PORT: 800, IDXGRP: 16#4020, IDXOFFS: 300, LEN: #4, SRCADDR: #5, WRITE: #10, TMOUT: timeout)
#7 SIZEOF(data_derevo)
#8 ADR(data_derevo)
#9 fb_floor4ADSwrite:ADSWRITE(NETID: ads_adr4, PORT: 800, IDXGRP: 16#4020, IDXOFFS: 0, LEN: #7, SRCADDR: #8, WRITE: MAIN.write4, TMOUT: timeout)
#10 OR(MAIN.write2, NOT heartbeat.Q)
#11 OR(MAIN.write1, NOT heartbeat.Q)
_END_CFC_
(* the same logic as Structured Text *)
fb_floor1ADSwrite(NETID := ads_adr1, PORT := 800, IDXGRP := 16#4020, IDXOFFS := 300, LEN := SIZEOF(data1floor), SRCADDR := ADR(data1floor), WRITE := _t99, TMOUT := timeout);
heartbeat(IN := NOT heartbeat.Q, PT := t#10s);
fb_floor2ADSwrite(NETID := ads_adr2, PORT := 800, IDXGRP := 16#4020, IDXOFFS := 300, LEN := SIZEOF(data2floor), SRCADDR := ADR(data2floor), WRITE := _t96, TMOUT := timeout);
fb_floor4ADSwrite(NETID := ads_adr4, PORT := 800, IDXGRP := 16#4020, IDXOFFS := 0, LEN := SIZEOF(data_derevo), SRCADDR := ADR(data_derevo), WRITE := MAIN.write4, TMOUT := timeout);
_t96 := MAIN.write2 OR NOT heartbeat.Q;
_t99 := MAIN.write1 OR NOT heartbeat.Q;
END_PROGRAM

(* POU HVAC/summer, ST *)
PROGRAM summer
VAR

END_VAR
data1floor[0].3:=heating_mode;

(*--------------------------VITALNYA---------------------------------------------------------------*)

	IF VITALNYA_HVAC.heat_mode=2 THEN (*heat*)
		IF heating_mode THEN VITALNYA_HVAC.zaslinka:=TRUE;(*closed*) ELSE VITALNYA_HVAC.zaslinka:=FALSE; (*opened*)END_IF;
		VITALNYA_HVAC.floor_heating:=TRUE; (*all opened*);
		CASE VITALNYA_HVAC.heat_speed OF
			1:	VITALNYA_HVAC.fancoil_speed:=1;
				IF NOT heating_mode THEN  VITALNYA_HVAC.klapan:=16#0; ELSE VITALNYA_HVAC.klapan:=16#3FFF;END_IF
			2:	VITALNYA_HVAC.fancoil_speed:=2;
				IF NOT heating_mode THEN  VITALNYA_HVAC.klapan:=16#0; ELSE VITALNYA_HVAC.klapan:=16#5FFF;END_IF
			3:	VITALNYA_HVAC.fancoil_speed:=3;
				IF NOT heating_mode THEN  VITALNYA_HVAC.klapan:=16#0; ELSE VITALNYA_HVAC.klapan:=16#7FFF;END_IF
		END_CASE
	END_IF

	IF VITALNYA_HVAC.heat_mode=1 THEN (*cool*)
		IF  heating_mode THEN VITALNYA_HVAC.klapan:=16#0;(*full closed*) END_IF
		IF  heating_mode THEN VITALNYA_HVAC.zaslinka:=FALSE; ELSE VITALNYA_HVAC.zaslinka:=TRUE; END_IF
				VITALNYA_HVAC.floor_heating:=FALSE; (*all closed*)

			CASE VITALNYA_HVAC.heat_speed OF
			1:	VITALNYA_HVAC.fancoil_speed:=1;
				IF NOT heating_mode THEN  VITALNYA_HVAC.klapan:=16#3FFF; ELSE VITALNYA_HVAC.klapan:=16#0;END_IF
			2:	VITALNYA_HVAC.fancoil_speed:=2;
				IF NOT heating_mode THEN  VITALNYA_HVAC.klapan:=16#5FFF; ELSE VITALNYA_HVAC.klapan:=16#0;END_IF
			3:	VITALNYA_HVAC.fancoil_speed:=3;
				IF NOT heating_mode THEN  VITALNYA_HVAC.klapan:=16#7FFF; ELSE VITALNYA_HVAC.klapan:=16#0;END_IF
		END_CASE
	END_IF

	IF VITALNYA_HVAC.heat_mode=3 THEN (*fan*)
		VITALNYA_HVAC.floor_heating:=FALSE;

		CASE VITALNYA_HVAC.heat_speed OF
			1:	VITALNYA_HVAC.fancoil_speed:=0;
				VITALNYA_HVAC.zaslinka:=TRUE;(*closed*)
				VITALNYA_HVAC.klapan:=16#0;(*full closed*)
			2:	VITALNYA_HVAC.fancoil_speed:=2;
				VITALNYA_HVAC.zaslinka:=FALSE;(*opened*)
				VITALNYA_HVAC.klapan:=16#7FFF;
			3:	VITALNYA_HVAC.fancoil_speed:=3;
				VITALNYA_HVAC.zaslinka:=FALSE;(*opened*)
				VITALNYA_HVAC.klapan:=16#7FFF;
		END_CASE
	IF t_out<0 THEN VITALNYA_HVAC.klapan:=16#5FFF; ELSE VITALNYA_HVAC.klapan:=16#0;END_IF
	END_IF



(*--------------------------KABINET---------------------------------------------------------------*)
(*реверс двигуна клапана*)

	IF kabinet_HVAC.heat_mode=2 THEN (*heat*)
		IF heating_mode THEN kabinet_HVAC.zaslinka:=TRUE;(*closed*) ELSE kabinet_HVAC.zaslinka:=FALSE; (*opened*)END_IF;
		kabinet_HVAC.floor_heating:=TRUE; (*all opened*);
		CASE kabinet_HVAC.heat_speed OF
			1:	kabinet_HVAC.fancoil_speed:=1;
				IF heating_mode THEN  kabinet_HVAC.klapan:=16#0; ELSE kabinet_HVAC.klapan:=16#7FFF;END_IF
			2:	kabinet_HVAC.fancoil_speed:=2;
				IF heating_mode THEN  kabinet_HVAC.klapan:=16#0; ELSE kabinet_HVAC.klapan:=16#5FFF;END_IF
			3:	kabinet_HVAC.fancoil_speed:=3;
				IF heating_mode THEN  kabinet_HVAC.klapan:=16#0; ELSE kabinet_HVAC.klapan:=16#3FFF;END_IF
		END_CASE
	END_IF

	IF kabinet_HVAC.heat_mode=1 THEN (*cool*)
		IF NOT heating_mode THEN kabinet_HVAC.klapan:=16#0;(*full closed*) END_IF
		IF NOT heating_mode THEN kabinet_HVAC.zaslinka:=FALSE; ELSE kabinet_HVAC.zaslinka:=TRUE; END_IF
				kabinet_HVAC.floor_heating:=FALSE; (*all closed*)

			CASE kabinet_HVAC.heat_speed OF
			1:	kabinet_HVAC.fancoil_speed:=1;
				IF heating_mode THEN  kabinet_HVAC.klapan:=16#7FFF; ELSE kabinet_HVAC.klapan:=16#0;END_IF
			2:	kabinet_HVAC.fancoil_speed:=2;
				IF heating_mode THEN  kabinet_HVAC.klapan:=16#5FFF; ELSE kabinet_HVAC.klapan:=16#0;END_IF
			3:	kabinet_HVAC.fancoil_speed:=3;
				IF heating_mode THEN  kabinet_HVAC.klapan:=16#3FFF; ELSE kabinet_HVAC.klapan:=16#0;END_IF
		END_CASE
	END_IF

	IF kabinet_HVAC.heat_mode=3 THEN (*fan*)
		kabinet_HVAC.floor_heating:=FALSE;
		IF t_out<0 THEN kabinet_HVAC.klapan:=16#3FFF;(*30%*) ELSE kabinet_HVAC.klapan:=16#0;END_IF
		CASE kabinet_HVAC.heat_speed OF
			1:	kabinet_HVAC.fancoil_speed:=0;
				kabinet_HVAC.zaslinka:=TRUE;(*closed*)
				kabinet_HVAC.klapan:=16#0;(*full closed*)
			2:	kabinet_HVAC.fancoil_speed:=2;
				kabinet_HVAC.zaslinka:=FALSE;(*opened*)
				kabinet_HVAC.klapan:=16#7FFF;
			3:	kabinet_HVAC.fancoil_speed:=3;
				kabinet_HVAC.zaslinka:=FALSE;(*opened*)
				kabinet_HVAC.klapan:=16#7FFF;
		END_CASE
	END_IF


(*--------------------------KINO---------------------------------------------------------------*)
(*реверс двигуна клапана*)

	IF KINO_HVAC.heat_mode=2 THEN (*heat*)
		IF heating_mode THEN KINO_HVAC.zaslinka:=TRUE;(*closed*) ELSE KINO_HVAC.zaslinka:=FALSE; (*opened*)END_IF;
		KINO_HVAC.floor_heating:=TRUE; (*all opened*);
		CASE KINO_HVAC.heat_speed OF
			1:	KINO_HVAC.fancoil_speed:=1;
				IF NOT heating_mode THEN  KINO_HVAC.klapan:=16#0; ELSE KINO_HVAC.klapan:=16#5FFF;END_IF
			2:	KINO_HVAC.fancoil_speed:=2;
				IF NOT heating_mode THEN  KINO_HVAC.klapan:=16#0; ELSE KINO_HVAC.klapan:=16#3FFF;END_IF
			3:	KINO_HVAC.fancoil_speed:=3;
				IF NOT heating_mode THEN  KINO_HVAC.klapan:=16#0; ELSE KINO_HVAC.klapan:=16#0;END_IF
		END_CASE
	END_IF

	IF KINO_HVAC.heat_mode=1 THEN (*cool*)
		IF  heating_mode THEN KINO_HVAC.klapan:=16#7FFF;(*full closed*) END_IF
		IF  heating_mode THEN KINO_HVAC.zaslinka:=FALSE; ELSE KINO_HVAC.zaslinka:=TRUE; END_IF
				KINO_HVAC.floor_heating:=FALSE; (*all closed*)

			CASE KINO_HVAC.heat_speed OF
			1:	KINO_HVAC.fancoil_speed:=1;
				IF NOT heating_mode THEN  KINO_HVAC.klapan:=16#5FFF; ELSE KINO_HVAC.klapan:=16#7FFF;END_IF
			2:	KINO_HVAC.fancoil_speed:=2;
				IF NOT heating_mode THEN  KINO_HVAC.klapan:=16#3FFF; ELSE KINO_HVAC.klapan:=16#7FFF;END_IF
			3:	KINO_HVAC.fancoil_speed:=3;
				IF NOT heating_mode THEN  KINO_HVAC.klapan:=16#0; ELSE KINO_HVAC.klapan:=16#7FFF;END_IF
		END_CASE
	END_IF

	IF KINO_HVAC.heat_mode=3 THEN (*fan*)
		KINO_HVAC.floor_heating:=FALSE;

		CASE KINO_HVAC.heat_speed OF
			1:	KINO_HVAC.fancoil_speed:=0;
				KINO_HVAC.zaslinka:=TRUE;(*closed*)
				KINO_HVAC.klapan:=16#7FFF;(*full closed*)
			2:	KINO_HVAC.fancoil_speed:=2;
				KINO_HVAC.zaslinka:=FALSE;(*opened*)
				KINO_HVAC.klapan:=16#7FFF;
			3:	KINO_HVAC.fancoil_speed:=3;
				KINO_HVAC.zaslinka:=FALSE;(*opened*)
				KINO_HVAC.klapan:=16#7FFF;
		END_CASE
		IF t_out<0 THEN KINO_HVAC.klapan:=16#5FFF;  ELSE KINO_HVAC.klapan:=16#7FFF;END_IF
	END_IF

(*--------------------------DYTJACHA---------------------------------------------------------------*)
(*реверс двигуна клапана*)

	IF dytjacha_HVAC.heat_mode=2 THEN (*heat*)
		IF heating_mode THEN dytjacha_HVAC.zaslinka:=TRUE;(*closed*) ELSE dytjacha_HVAC.zaslinka:=FALSE; (*opened*)END_IF;
		dytjacha_HVAC.floor_heating:=TRUE; (*all opened*);
		CASE dytjacha_HVAC.heat_speed OF
			1:	dytjacha_HVAC.fancoil_speed:=1;
				IF NOT heating_mode THEN  dytjacha_HVAC.klapan:=16#7FFF; ELSE dytjacha_HVAC.klapan:=16#5FFF;END_IF
			2:	dytjacha_HVAC.fancoil_speed:=2;
				IF NOT heating_mode THEN  dytjacha_HVAC.klapan:=16#7FFF; ELSE dytjacha_HVAC.klapan:=16#3FFF;END_IF
			3:	dytjacha_HVAC.fancoil_speed:=3;
				IF NOT heating_mode THEN  dytjacha_HVAC.klapan:=16#7FFF; ELSE dytjacha_HVAC.klapan:=16#0;END_IF
		END_CASE
	END_IF

	IF dytjacha_HVAC.heat_mode=1 THEN (*cool*)
		IF  heating_mode THEN dytjacha_HVAC.klapan:=16#7FFF;(*full closed*) END_IF
		IF  heating_mode THEN dytjacha_HVAC.zaslinka:=FALSE; ELSE dytjacha_HVAC.zaslinka:=TRUE; END_IF
				dytjacha_HVAC.floor_heating:=FALSE; (*all closed*)

			CASE dytjacha_HVAC.heat_speed OF
			1:	dytjacha_HVAC.fancoil_speed:=1;
				IF heating_mode THEN  dytjacha_HVAC.klapan:=16#7FFF; ELSE dytjacha_HVAC.klapan:=16#0;END_IF
			2:	dytjacha_HVAC.fancoil_speed:=2;
				IF heating_mode THEN  dytjacha_HVAC.klapan:=16#5FFF; ELSE dytjacha_HVAC.klapan:=16#0;END_IF
			3:	dytjacha_HVAC.fancoil_speed:=3;
				IF heating_mode THEN  dytjacha_HVAC.klapan:=16#3FFF; ELSE dytjacha_HVAC.klapan:=16#0;END_IF
		END_CASE
	END_IF

	IF dytjacha_HVAC.heat_mode=3 THEN (*fan*)
		dytjacha_HVAC.floor_heating:=FALSE;
		CASE dytjacha_HVAC.heat_speed OF
			1:	dytjacha_HVAC.fancoil_speed:=0;
				dytjacha_HVAC.zaslinka:=TRUE;(*closed*)
				dytjacha_HVAC.klapan:=16#0;(*full closed*)
			2:	dytjacha_HVAC.fancoil_speed:=2;
				dytjacha_HVAC.zaslinka:=FALSE;(*opened*)
				dytjacha_HVAC.klapan:=16#7FFF;
			3:	dytjacha_HVAC.fancoil_speed:=3;
				dytjacha_HVAC.zaslinka:=FALSE;(*opened*)
				dytjacha_HVAC.klapan:=16#7FFF;
		END_CASE
		IF t_out<0 THEN dytjacha_HVAC.klapan:=16#5FFF; ELSE dytjacha_HVAC.klapan:=16#7FFF;END_IF
	END_IF
(*--------------------------SPALNYA---------------------------------------------------------------*)

	IF SPALNYA_HVAC.heat_mode=2 THEN (*heat*)
		IF heating_mode THEN SPALNYA_HVAC.zaslinka:=TRUE;(*closed*) ELSE SPALNYA_HVAC.zaslinka:=FALSE; (*opened*)END_IF;
		SPALNYA_HVAC.floor_heating:=TRUE; (*all opened*);
		CASE SPALNYA_HVAC.heat_speed OF
			1:	SPALNYA_HVAC.fancoil_speed:=1;
				IF NOT  heating_mode THEN  SPALNYA_HVAC.klapan:=16#0; ELSE SPALNYA_HVAC.klapan:=16#3FFF;END_IF
			2:	SPALNYA_HVAC.fancoil_speed:=2;
				IF NOT heating_mode THEN  SPALNYA_HVAC.klapan:=16#0; ELSE SPALNYA_HVAC.klapan:=16#5FFF;END_IF
			3:	SPALNYA_HVAC.fancoil_speed:=3;
				IF NOT heating_mode THEN  SPALNYA_HVAC.klapan:=16#0; ELSE SPALNYA_HVAC.klapan:=16#7FFF;END_IF
		END_CASE
	END_IF

	IF SPALNYA_HVAC.heat_mode=1 THEN (*cool*)
		IF  heating_mode THEN SPALNYA_HVAC.klapan:=16#5FFF;(*full closed*) END_IF
		IF  heating_mode THEN SPALNYA_HVAC.zaslinka:=FALSE; ELSE SPALNYA_HVAC.zaslinka:=TRUE; END_IF
				SPALNYA_HVAC.floor_heating:=FALSE; (*all closed*)

			CASE SPALNYA_HVAC.heat_speed OF
			1:	SPALNYA_HVAC.fancoil_speed:=1;
				IF NOT heating_mode THEN  SPALNYA_HVAC.klapan:=16#3FFF; ELSE SPALNYA_HVAC.klapan:=16#0;END_IF
			2:	SPALNYA_HVAC.fancoil_speed:=2;
				IF NOT heating_mode THEN  SPALNYA_HVAC.klapan:=16#5FFF; ELSE SPALNYA_HVAC.klapan:=16#0;END_IF
			3:	SPALNYA_HVAC.fancoil_speed:=3;
				IF NOT heating_mode THEN  SPALNYA_HVAC.klapan:=16#7FFF; ELSE SPALNYA_HVAC.klapan:=16#0;END_IF
		END_CASE
	END_IF

	IF SPALNYA_HVAC.heat_mode=3 THEN (*fan*)
		SPALNYA_HVAC.floor_heating:=FALSE;
		CASE SPALNYA_HVAC.heat_speed OF
			1:	SPALNYA_HVAC.fancoil_speed:=0;
				SPALNYA_HVAC.zaslinka:=TRUE;(*closed*)
				SPALNYA_HVAC.klapan:=16#0;(*full closed*)
			2:	SPALNYA_HVAC.fancoil_speed:=2;
				SPALNYA_HVAC.zaslinka:=FALSE;(*opened*)
				SPALNYA_HVAC.klapan:=16#0;
			3:	SPALNYA_HVAC.fancoil_speed:=3;
				SPALNYA_HVAC.zaslinka:=FALSE;(*opened*)
				SPALNYA_HVAC.klapan:=16#0;
		END_CASE
		IF t_out<0 THEN SPALNYA_HVAC.klapan:=16#3FFF;(*30%*) ELSE SPALNYA_HVAC.klapan:=16#0;END_IF
	END_IF
END_PROGRAM

(* POU HVAC/winter, ST *)
PROGRAM winter
VAR

END_VAR
(*1-COOL mode 2-HEAT mode, 3-FAN mode*)

(*--------------------------VITALNYA---------------------------------------------------------------*)

	IF VITALNYA_HVAC.heat_mode=2 THEN
				VITALNYA_HVAC.zaslinka:=TRUE;(*closed*)
				VITALNYA_HVAC.floor_heating:=TRUE; (*all opened*)
		CASE VITALNYA_HVAC.heat_speed OF

			1:	VITALNYA_HVAC.fancoil_speed:=1;
				VITALNYA_HVAC.klapan:=16#3FFF;
			2:	VITALNYA_HVAC.fancoil_speed:=2;
				VITALNYA_HVAC.klapan:=16#5FFF;
			3:	VITALNYA_HVAC.fancoil_speed:=3;
				VITALNYA_HVAC.klapan:=16#7FFF;
		END_CASE
	END_IF

	IF VITALNYA_HVAC.heat_mode=1 THEN
				VITALNYA_HVAC.klapan:=16#0;(*full closed*)
				VITALNYA_HVAC.zaslinka:=FALSE;
				VITALNYA_HVAC.floor_heating:=FALSE; (*all closed*)

			CASE VITALNYA_HVAC.heat_speed OF
			1:	VITALNYA_HVAC.fancoil_speed:=1;
			2:	VITALNYA_HVAC.fancoil_speed:=2;
			3:	VITALNYA_HVAC.fancoil_speed:=3;
		END_CASE
	END_IF

	IF VITALNYA_HVAC.heat_mode=3 THEN
		VITALNYA_HVAC.floor_heating:=FALSE;
		IF t_out<0 THEN VITALNYA_HVAC.klapan:=16#3FFF;(*30%*) ELSE VITALNYA_HVAC.klapan:=16#0;END_IF
		CASE VITALNYA_HVAC.heat_speed OF
			1:	VITALNYA_HVAC.fancoil_speed:=0;
				VITALNYA_HVAC.zaslinka:=TRUE;(*closed*)
				VITALNYA_HVAC.klapan:=16#0;(*full closed*)
			2:	VITALNYA_HVAC.fancoil_speed:=2;
				VITALNYA_HVAC.zaslinka:=FALSE;(*opened*)
			3:	VITALNYA_HVAC.fancoil_speed:=3;
				VITALNYA_HVAC.zaslinka:=FALSE;(*opened*)
		END_CASE
	END_IF



(*--------------------------KABINET---------------------------------------------------------------*)
(*реверс двигуна клапана*)

	IF KABINET_HVAC.heat_mode=2 THEN
				KABINET_HVAC.zaslinka:=TRUE;(*closed*)
				KABINET_HVAC.floor_heating:=TRUE; (*all opened*)
		CASE KABINET_HVAC.heat_speed OF

			1:	KABINET_HVAC.fancoil_speed:=1;
				KABINET_HVAC.klapan:=16#5FFF;
			2:	KABINET_HVAC.fancoil_speed:=2;
				KABINET_HVAC.klapan:=16#3FFF;
			3:	KABINET_HVAC.fancoil_speed:=3;
				KABINET_HVAC.klapan:=16#1FFF;
		END_CASE
	END_IF

	IF KABINET_HVAC.heat_mode=1 THEN
				KABINET_HVAC.klapan:=16#7FFF;(*full closed*)
				KABINET_HVAC.zaslinka:=FALSE;
				KABINET_HVAC.floor_heating:=FALSE; (*all closed*)

			CASE KABINET_HVAC.heat_speed OF
			1:	KABINET_HVAC.fancoil_speed:=1;
			2:	KABINET_HVAC.fancoil_speed:=2;
			3:	KABINET_HVAC.fancoil_speed:=3;
		END_CASE
	END_IF

	IF KABINET_HVAC.heat_mode=3 THEN
		KABINET_HVAC.floor_heating:=FALSE;
		IF t_out<0 THEN KABINET_HVAC.klapan:=16#5FFF;(*30%*) ELSE KABINET_HVAC.klapan:=16#7FFF;END_IF
		CASE KABINET_HVAC.heat_speed OF
			1:	KABINET_HVAC.fancoil_speed:=0;
				KABINET_HVAC.zaslinka:=TRUE;(*closed*)
				KABINET_HVAC.klapan:=16#7FFF;(*full closed*)
			2:	KABINET_HVAC.fancoil_speed:=2;
				KABINET_HVAC.zaslinka:=FALSE;(*opened*)
			3:	KABINET_HVAC.fancoil_speed:=3;
				KABINET_HVAC.zaslinka:=FALSE;(*opened*)
		END_CASE
	END_IF



(*--------------------------KINO---------------------------------------------------------------*)
(*реверс двигуна клапана*)
	IF KINO_HVAC.heat_mode=2 THEN
				KINO_HVAC.zaslinka:=TRUE;(*closed*)
				KINO_HVAC.floor_heating:=TRUE; (*all opened*)
		CASE KINO_HVAC.heat_speed OF

			1:	KINO_HVAC.fancoil_speed:=1;
				KINO_HVAC.klapan:=16#5FFF;
			2:	KINO_HVAC.fancoil_speed:=2;
				KINO_HVAC.klapan:=16#3FFF;
			3:	KINO_HVAC.fancoil_speed:=3;
				KINO_HVAC.klapan:=16#1FFF;
		END_CASE
	END_IF

	IF KINO_HVAC.heat_mode=1 THEN
				KINO_HVAC.klapan:=16#0;(*full closed*)
				KINO_HVAC.zaslinka:=FALSE;
				KINO_HVAC.floor_heating:=FALSE; (*all closed*)

			CASE KINO_HVAC.heat_speed OF
			1:	KINO_HVAC.fancoil_speed:=1;
			2:	KINO_HVAC.fancoil_speed:=2;
			3:	KINO_HVAC.fancoil_speed:=3;
		END_CASE
	END_IF

	IF KINO_HVAC.heat_mode=3 THEN
		KINO_HVAC.floor_heating:=FALSE;
		IF t_out<0 THEN KINO_HVAC.klapan:=16#5FFF;(*30%*) ELSE KINO_HVAC.klapan:=16#7FFF;END_IF
		CASE KINO_HVAC.heat_speed OF
			1:	KINO_HVAC.fancoil_speed:=0;
				KINO_HVAC.zaslinka:=TRUE;(*closed*)
				KINO_HVAC.klapan:=16#7FFF;(*full closed*)
			2:	KINO_HVAC.fancoil_speed:=2;
				KINO_HVAC.zaslinka:=FALSE;(*opened*)
			3:	KINO_HVAC.fancoil_speed:=3;
				KINO_HVAC.zaslinka:=FALSE;(*opened*)
		END_CASE
	END_IF



(*--------------------------DYTJACHA---------------------------------------------------------------*)
(*реверс двигуна клапана*)
	IF DYTJACHA_HVAC.heat_mode=2 THEN
				DYTJACHA_HVAC.zaslinka:=TRUE;(*closed*)
				DYTJACHA_HVAC.floor_heating:=TRUE; (*all opened*)
		CASE DYTJACHA_HVAC.heat_speed OF

			1:	DYTJACHA_HVAC.fancoil_speed:=1;
				DYTJACHA_HVAC.klapan:=16#5FFF;
			2:	DYTJACHA_HVAC.fancoil_speed:=2;
				DYTJACHA_HVAC.klapan:=16#3FFF;
			3:	DYTJACHA_HVAC.fancoil_speed:=3;
				DYTJACHA_HVAC.klapan:=16#1FFF;
		END_CASE
	END_IF

	IF DYTJACHA_HVAC.heat_mode=1 THEN
				DYTJACHA_HVAC.klapan:=16#7FFF;(*full closed*)
				DYTJACHA_HVAC.zaslinka:=FALSE;
				DYTJACHA_HVAC.floor_heating:=FALSE; (*all closed*)

			CASE DYTJACHA_HVAC.heat_speed OF
			1:	DYTJACHA_HVAC.fancoil_speed:=1;
			2:	DYTJACHA_HVAC.fancoil_speed:=2;
			3:	DYTJACHA_HVAC.fancoil_speed:=3;
		END_CASE
	END_IF

	IF DYTJACHA_HVAC.heat_mode=3 THEN
		DYTJACHA_HVAC.floor_heating:=FALSE;
		IF t_out<0 THEN DYTJACHA_HVAC.klapan:=16#5FFF;(*30%*) ELSE DYTJACHA_HVAC.klapan:=16#7FFF;END_IF
		CASE DYTJACHA_HVAC.heat_speed OF
			1:	DYTJACHA_HVAC.fancoil_speed:=0;
				DYTJACHA_HVAC.zaslinka:=TRUE;(*closed*)
				DYTJACHA_HVAC.klapan:=16#7FFF;(*full closed*)
			2:	DYTJACHA_HVAC.fancoil_speed:=2;
				DYTJACHA_HVAC.zaslinka:=FALSE;(*opened*)
			3:	DYTJACHA_HVAC.fancoil_speed:=3;
				DYTJACHA_HVAC.zaslinka:=FALSE;(*opened*)
		END_CASE
	END_IF



(*--------------------------SPALNYA---------------------------------------------------------------*)

	IF SPALNYA_HVAC.heat_mode=2 THEN
				SPALNYA_HVAC.zaslinka:=TRUE;(*closed*)
				SPALNYA_HVAC.floor_heating:=TRUE; (*all opened*)
		CASE SPALNYA_HVAC.heat_speed OF

			1:	SPALNYA_HVAC.fancoil_speed:=1;
				SPALNYA_HVAC.klapan:=16#3FFF;
			2:	SPALNYA_HVAC.fancoil_speed:=2;
				SPALNYA_HVAC.klapan:=16#5FFF;
			3:	SPALNYA_HVAC.fancoil_speed:=3;
				SPALNYA_HVAC.klapan:=16#7FFF;
		END_CASE
	END_IF

	IF SPALNYA_HVAC.heat_mode=1 THEN
				SPALNYA_HVAC.klapan:=16#0;(*full closed*)
				SPALNYA_HVAC.zaslinka:=FALSE;
				SPALNYA_HVAC.floor_heating:=FALSE; (*all closed*)

			CASE SPALNYA_HVAC.heat_speed OF
			1:	SPALNYA_HVAC.fancoil_speed:=1;
			2:	SPALNYA_HVAC.fancoil_speed:=2;
			3:	SPALNYA_HVAC.fancoil_speed:=3;
		END_CASE
	END_IF

	IF SPALNYA_HVAC.heat_mode=3 THEN
		SPALNYA_HVAC.floor_heating:=FALSE;
		IF t_out<0 THEN SPALNYA_HVAC.klapan:=16#3FFF;(*30%*) ELSE SPALNYA_HVAC.klapan:=16#0;END_IF
		CASE SPALNYA_HVAC.heat_speed OF
			1:	SPALNYA_HVAC.fancoil_speed:=0;
				SPALNYA_HVAC.zaslinka:=TRUE;(*closed*)
				SPALNYA_HVAC.klapan:=16#0;(*full closed*)
			2:	SPALNYA_HVAC.fancoil_speed:=2;
				SPALNYA_HVAC.zaslinka:=FALSE;(*opened*)
			3:	SPALNYA_HVAC.fancoil_speed:=3;
				SPALNYA_HVAC.zaslinka:=FALSE;(*opened*)
		END_CASE
	END_IF
END_PROGRAM

(* POU Vymykachi/SWITCH, ST *)
FUNCTION_BLOCK SWITCH
VAR_INPUT
	IN:BOOL;
	SHORT_OFF_DELAY, LONG_OFF_DELAY: TIME; (*час затримки вимкнення по короткому та довгому натисненню*)
END_VAR
VAR_OUTPUT
	short, long:BOOL;
END_VAR
VAR
	tChas: TIME; (*час доки кнопка натиснена*)
	TIMER: TON; (*таймер час натискання*)
	bPressed:BOOL;
	turn_off_long: BOOL;
	start_l, start_s:BOOL;
	bStan: BOOL:=FALSE;
END_VAR
short:=FALSE;
long:=FALSE;
TIMER(IN:=IN AND bStan, PT:=t#10s);
IF IN AND bStan THEN
	tChas:=timer.ET;
	bPressed:=TRUE;
ELSE
	bPressed:=FALSE;
END_IF;

IF NOT IN AND NOT bStan THEN
	tChas:=t#0ms;
END_IF;

IF bStan AND NOT IN THEN
	IF tChas <tLongPress THEN
		short:=TRUE;
	END_IF;
	IF tChas>=tLongPress THEN
		long:=TRUE;
	END_IF;
END_IF;
bStan := IN;
END_FUNCTION_BLOCK
